   VAR_IN_OUT 
      xNewRecord { ExternalAccessible := 'False'; ExternalVisible := 'False'; ExternalWritable := 'False'} : Bool;
      xProductionRecord { ExternalAccessible := 'False'; ExternalVisible := 'False'; ExternalWritable := 'False'} : Bool;
      xLeftRobotUsed { ExternalAccessible := 'False'; ExternalVisible := 'False'; ExternalWritable := 'False'} : Bool;
      xRightRobotUsed { ExternalAccessible := 'False'; ExternalVisible := 'False'; ExternalWritable := 'False'} : Bool;
      xResetCurrentRecord { ExternalAccessible := 'False'; ExternalVisible := 'False'; ExternalWritable := 'False'} : Bool;
      xEraseAllData { ExternalAccessible := 'False'; ExternalVisible := 'False'; ExternalWritable := 'False'} : Bool;
      xDisplayNextRecord { ExternalAccessible := 'False'; ExternalVisible := 'False'; ExternalWritable := 'False'} : Bool;
      xDisplayPrevRecord { ExternalAccessible := 'False'; ExternalVisible := 'False'; ExternalWritable := 'False'} : Bool;
      uiNumberOfRecords { ExternalAccessible := 'False'; ExternalVisible := 'False'; ExternalWritable := 'False'} : UInt;
      aProdData : Array[*] of "stProductionRecord";
   END_VAR

   VAR 
      sxNewRecord { ExternalAccessible := 'False'; ExternalVisible := 'False'; ExternalWritable := 'False'} : Bool;
      sdiMaxRecord { ExternalAccessible := 'False'; ExternalVisible := 'False'; ExternalWritable := 'False'} : DInt;
      snCounter { ExternalAccessible := 'False'; ExternalVisible := 'False'; ExternalWritable := 'False'} : Int;
      suiMemDisplayCurentReccord { ExternalAccessible := 'False'; ExternalVisible := 'False'; ExternalWritable := 'False'} : UInt;
      suiMaxJobNumber { ExternalAccessible := 'False'; ExternalVisible := 'False'; ExternalWritable := 'False'} : UInt;
      suiMemCurrentJobNumberR1 { ExternalAccessible := 'False'; ExternalVisible := 'False'; ExternalWritable := 'False'} : UInt;
      suiMemCurrentJobNumberR2 { ExternalAccessible := 'False'; ExternalVisible := 'False'; ExternalWritable := 'False'} : UInt;
      suiDisplayCurentRecord { ExternalAccessible := 'False'; ExternalVisible := 'False'; ExternalWritable := 'False'} : UInt;
   END_VAR

   VAR_TEMP 
      txRequestAction : Bool;
      suiCount : UInt;
      suiRecord : UInt;
      tuiPaperUsedRobot1 : UInt;
      tuiPaperUsedRobot2 : UInt;
   END_VAR


BEGIN
	REGION Control Job Number Used
	  // Control if record data is in pregress and Job Data number change
	  IF #sxNewRecord AND (#uiCurrentJobNumberRobot1 <> #suiMemCurrentJobNumberR1) THEN
	    // Controo if job data number is in range
	    IF ((#uiCurrentJobNumberRobot1 > 0) AND (#uiCurrentJobNumberRobot1 <= 6)) THEN
	      #suiMemCurrentJobNumberR1 := #uiCurrentJobNumberRobot1;
	      CASE #uiCurrentJobNumberRobot1 OF
	        1:
	          #aProdData[1].Rob1Job1Used := TRUE;
	          #aProdData[1].Rob1Job1DistChangePaper := #WorkRecipe.RecipeLayerType.JobTableLeft[1].WornPaperDistance;
	          #aProdData[1].Rob1Job1ForceTarget := #WorkRecipe.RecipeLayerType.JobTableLeft[1].SetForceTarget;
	          #aProdData[1].Rob1Job1RobotSpeed := #WorkRecipe.RecipeLayerType.JobTableLeft[1].SetRobotSpeed;
	          #aProdData[1].Rob1Job1SandingSpeed := #WorkRecipe.RecipeLayerType.JobTableLeft[1].SetSpeed;
	        2:
	          #aProdData[1].Rob1Job2Used := TRUE;
	          #aProdData[1].Rob1Job2DistChangePaper := #WorkRecipe.RecipeLayerType.JobTableLeft[2].WornPaperDistance;
	          #aProdData[1].Rob1Job2ForceTarget := #WorkRecipe.RecipeLayerType.JobTableLeft[2].SetForceTarget;
	          #aProdData[1].Rob1Job2RobotSpeed := #WorkRecipe.RecipeLayerType.JobTableLeft[2].SetRobotSpeed;
	          #aProdData[1].Rob1Job2SandingSpeed := #WorkRecipe.RecipeLayerType.JobTableLeft[2].SetSpeed;
	        3:
	          #aProdData[1].Rob1Job3Used := TRUE;
	          #aProdData[1].Rob1Job3DistChangePaper := #WorkRecipe.RecipeLayerType.JobTableLeft[3].WornPaperDistance;
	          #aProdData[1].Rob1Job3ForceTarget := #WorkRecipe.RecipeLayerType.JobTableLeft[3].SetForceTarget;
	          #aProdData[1].Rob1Job3RobotSpeed := #WorkRecipe.RecipeLayerType.JobTableLeft[3].SetRobotSpeed;
	          #aProdData[1].Rob1Job3SandingSpeed := #WorkRecipe.RecipeLayerType.JobTableLeft[3].SetSpeed;
	        4:
	          #aProdData[1].Rob1Job4Used := TRUE;
	          #aProdData[1].Rob1Job4DistChangePaper := #WorkRecipe.RecipeLayerType.JobTableLeft[4].WornPaperDistance;
	          #aProdData[1].Rob1Job4ForceTarget := #WorkRecipe.RecipeLayerType.JobTableLeft[4].SetForceTarget;
	          #aProdData[1].Rob1Job4RobotSpeed := #WorkRecipe.RecipeLayerType.JobTableLeft[4].SetRobotSpeed;
	          #aProdData[1].Rob1Job4SandingSpeed := #WorkRecipe.RecipeLayerType.JobTableLeft[4].SetSpeed;
	        5:
	          #aProdData[1].Rob1Job5Used := TRUE;
	          #aProdData[1].Rob1Job5DistChangePaper := #WorkRecipe.RecipeLayerType.JobTableLeft[5].WornPaperDistance;
	          #aProdData[1].Rob1Job5ForceTarget := #WorkRecipe.RecipeLayerType.JobTableLeft[5].SetForceTarget;
	          #aProdData[1].Rob1Job5RobotSpeed := #WorkRecipe.RecipeLayerType.JobTableLeft[5].SetRobotSpeed;
	          #aProdData[1].Rob1Job5SandingSpeed := #WorkRecipe.RecipeLayerType.JobTableLeft[5].SetSpeed;
	        6:
	          #aProdData[1].Rob1Job6Used := TRUE;
	          #aProdData[1].Rob1Job6DistChangePaper := #WorkRecipe.RecipeLayerType.JobTableLeft[6].WornPaperDistance;
	          #aProdData[1].Rob1Job6ForceTarget := #WorkRecipe.RecipeLayerType.JobTableLeft[6].SetForceTarget;
	          #aProdData[1].Rob1Job6RobotSpeed := #WorkRecipe.RecipeLayerType.JobTableLeft[6].SetRobotSpeed;
	          #aProdData[1].Rob1Job6SandingSpeed := #WorkRecipe.RecipeLayerType.JobTableLeft[6].SetSpeed;
	      END_CASE;
	      
	    ELSE
	      #suiMemCurrentJobNumberR1 := #uiCurrentJobNumberRobot1;
	    END_IF;
	  END_IF;
	  
	  // Control if record data is in pregress and Job Data number change
	  IF #sxNewRecord AND (#uiCurrentJobNumberRobot2 <> #suiMemCurrentJobNumberR2) THEN
	    // Controo if job data number is in range
	    IF ((#uiCurrentJobNumberRobot2 > 0) AND (#uiCurrentJobNumberRobot2 <= 6)) THEN
	      #suiMemCurrentJobNumberR2 := #uiCurrentJobNumberRobot2;
	      CASE #uiCurrentJobNumberRobot2 OF
	        1:
	          #aProdData[1].Rob2Job1Used := TRUE;
	          #aProdData[1].Rob2Job1DistChangePaper := #WorkRecipe.RecipeLayerType.JobTableRight[1].WornPaperDistance;
	          #aProdData[1].Rob2Job1ForceTarget := #WorkRecipe.RecipeLayerType.JobTableRight[1].SetForceTarget;
	          #aProdData[1].Rob2Job1RobotSpeed := #WorkRecipe.RecipeLayerType.JobTableRight[1].SetRobotSpeed;
	          #aProdData[1].Rob2Job1SandingSpeed := #WorkRecipe.RecipeLayerType.JobTableRight[1].SetSpeed;
	        2:
	          #aProdData[1].Rob2Job2Used := TRUE;
	          #aProdData[1].Rob2Job2DistChangePaper := #WorkRecipe.RecipeLayerType.JobTableRight[2].WornPaperDistance;
	          #aProdData[1].Rob2Job2ForceTarget := #WorkRecipe.RecipeLayerType.JobTableRight[2].SetForceTarget;
	          #aProdData[1].Rob2Job2RobotSpeed := #WorkRecipe.RecipeLayerType.JobTableRight[2].SetRobotSpeed;
	          #aProdData[1].Rob2Job2SandingSpeed := #WorkRecipe.RecipeLayerType.JobTableRight[2].SetSpeed;
	        3:
	          #aProdData[1].Rob2Job3Used := TRUE;
	          #aProdData[1].Rob2Job3DistChangePaper := #WorkRecipe.RecipeLayerType.JobTableRight[3].WornPaperDistance;
	          #aProdData[1].Rob2Job3ForceTarget := #WorkRecipe.RecipeLayerType.JobTableRight[3].SetForceTarget;
	          #aProdData[1].Rob2Job3RobotSpeed := #WorkRecipe.RecipeLayerType.JobTableRight[3].SetRobotSpeed;
	          #aProdData[1].Rob2Job3SandingSpeed := #WorkRecipe.RecipeLayerType.JobTableRight[3].SetSpeed;
	        4:
	          #aProdData[1].Rob2Job4Used := TRUE;
	          #aProdData[1].Rob2Job4DistChangePaper := #WorkRecipe.RecipeLayerType.JobTableRight[4].WornPaperDistance;
	          #aProdData[1].Rob2Job4ForceTarget := #WorkRecipe.RecipeLayerType.JobTableRight[4].SetForceTarget;
	          #aProdData[1].Rob2Job4RobotSpeed := #WorkRecipe.RecipeLayerType.JobTableRight[4].SetRobotSpeed;
	          #aProdData[1].Rob2Job4SandingSpeed := #WorkRecipe.RecipeLayerType.JobTableRight[4].SetSpeed;
	        5:
	          #aProdData[1].Rob2Job5Used := TRUE;
	          #aProdData[1].Rob2Job5DistChangePaper := #WorkRecipe.RecipeLayerType.JobTableRight[5].WornPaperDistance;
	          #aProdData[1].Rob2Job5ForceTarget := #WorkRecipe.RecipeLayerType.JobTableRight[5].SetForceTarget;
	          #aProdData[1].Rob2Job5RobotSpeed := #WorkRecipe.RecipeLayerType.JobTableRight[5].SetRobotSpeed;
	          #aProdData[1].Rob2Job5SandingSpeed := #WorkRecipe.RecipeLayerType.JobTableRight[5].SetSpeed;
	        6:
	          #aProdData[1].Rob2Job6Used := TRUE;
	          #aProdData[1].Rob2Job6DistChangePaper := #WorkRecipe.RecipeLayerType.JobTableRight[6].WornPaperDistance;
	          #aProdData[1].Rob2Job6ForceTarget := #WorkRecipe.RecipeLayerType.JobTableRight[6].SetForceTarget;
	          #aProdData[1].Rob2Job6RobotSpeed := #WorkRecipe.RecipeLayerType.JobTableRight[6].SetRobotSpeed;
	          #aProdData[1].Rob2Job6SandingSpeed := #WorkRecipe.RecipeLayerType.JobTableRight[6].SetSpeed;
	      END_CASE;
	    ELSE
	      #suiMemCurrentJobNumberR2 := #uiCurrentJobNumberRobot2;
	    END_IF;
	  END_IF;
	END_REGION
	
	REGION Exit FB
	  // Exit function bloc if no action requested
	  IF #suiDisplayCurentRecord = 0 THEN
	    #suiDisplayCurentRecord := 1;
	  END_IF;
	  
	  #txRequestAction := #xNewRecord OR #xProductionRecord OR #xResetCurrentRecord OR #xEraseAllData OR #xDisplayNextRecord OR #xDisplayPrevRecord;
	  IF #suiDisplayCurentRecord <> #suiMemDisplayCurentReccord THEN
	    #suiMemDisplayCurentReccord := #suiDisplayCurentRecord;
	  ELSIF (NOT #txRequestAction) THEN
	    RETURN;
	  END_IF;
	END_REGION
	
	REGION Record Min and Max
	  #sdiMaxRecord := UPPER_BOUND(ARR := #aProdData, DIM := 1);
	  IF #uiNumberOfRecords < 1 THEN
	    #uiRecordMax := 1;
	  ELSE
	    #uiRecordMax := #uiNumberOfRecords;
	  END_IF;
	  #uiRecordMin := 1;
	END_REGION
	
	REGION New Record
	  IF #xNewRecord AND (NOT #sxNewRecord) THEN // Request new record and no new record in progress
	    IF #uiNumberOfRecords = 0 THEN // First record
	      // First record in the table
	      #uiNumberOfRecords := 1;
	      // Erase all data
	      #aProdData[1] := #aProdData[0];
	      "FC71_PrepareNewRecord"(usiCurrentLayerType:=#usiCurrentLayerType,
	                              uiCbsNumber:=#uiCbsNumber,
	                              WorkRecipe:=#WorkRecipe,
	                              ProdData:=#aProdData[1]);
	    ELSIF #uiNumberOfRecords < #sdiMaxRecord THEN // less then max record
	      // Increase the number of record
	      #uiNumberOfRecords += 1;
	      // Offset all records
	      FOR #snCounter := UINT_TO_INT(#uiNumberOfRecords) TO 2 BY -1 DO
	        #aProdData[#snCounter] := #aProdData[#snCounter - 1];
	      END_FOR;
	      // Erase all data
	      #aProdData[1] := #aProdData[0];
	      "FC71_PrepareNewRecord"(usiCurrentLayerType := #usiCurrentLayerType,
	                              uiCbsNumber := #uiCbsNumber,
	                              WorkRecipe := #WorkRecipe,
	                              ProdData := #aProdData[1]);
	    ELSIF #uiNumberOfRecords = #sdiMaxRecord THEN // Max record
	      // Delete last record
	      #aProdData[#uiNumberOfRecords] := #aProdData[0];
	      // Offset all records
	      FOR #snCounter := UINT_TO_INT(#uiNumberOfRecords) TO 2 BY -1 DO
	        #aProdData[#snCounter] := #aProdData[#snCounter - 1];
	      END_FOR;
	      // Erase all data
	      #aProdData[1] := #aProdData[0];
	      "FC71_PrepareNewRecord"(usiCurrentLayerType := #usiCurrentLayerType,
	                              uiCbsNumber := #uiCbsNumber,
	                              WorkRecipe := #WorkRecipe,
	                              ProdData := #aProdData[1]);
	    END_IF;
	    #xNewRecord := FALSE;
	    #sxNewRecord := TRUE;
	    
	  ELSIF #xNewRecord AND #sxNewRecord THEN // Request new record but new record already in progress
	    #xNewRecord := FALSE;
	  END_IF;
	END_REGION
	
	REGION Production Record
	  IF #xProductionRecord AND #sxNewRecord THEN // Request record production and new record already in progress
	    // Count paper used if robot 1 used
	    IF #xLeftRobotUsed THEN
	      #tuiPaperUsedRobot1 := #uiPaperUsedRobot1;
	      #xLeftRobotUsed := FALSE;
	    ELSE
	      #tuiPaperUsedRobot1 := 0;
	    END_IF;
	    // Count paper used if robot 2 used
	    IF #xRightRobotUsed THEN
	      #tuiPaperUsedRobot2 := #uiPaperUsedRobot2;
	      #xRightRobotUsed := FALSE;
	    ELSE
	      #tuiPaperUsedRobot2 := 0;
	    END_IF;
	    // General record
	    "FC72_Record"(uiPaperUsedRobot1:=#tuiPaperUsedRobot1,
	                  uiPaperUsedRobot2:=#tuiPaperUsedRobot2,
	                  ProdData:=#aProdData[1]);
	    
	    #xProductionRecord := FALSE;
	    #sxNewRecord := FALSE;
	    
	  ELSIF #xProductionRecord AND (NOT #sxNewRecord) THEN // Request record production but no new record already in progress
	    #xProductionRecord := FALSE;
	    
	  END_IF;
	END_REGION
	
	REGION Erase All
	  IF #xEraseAllData THEN // Request reset all record in the table
	    // Erase all the data record
	    FOR #snCounter := 1 TO UINT_TO_INT(#uiNumberOfRecords) DO
	      #aProdData[#snCounter] := #aProdData[0];
	    END_FOR;
	    // Reset the number of record in table
	    #suiDisplayCurentRecord := 1;
	    #uiNumberOfRecords := 0;
	    #sxNewRecord := FALSE;
	    #xEraseAllData := FALSE;
	  END_IF;
	END_REGION
	
	REGION Erase Record
	  IF #xResetCurrentRecord AND #sxNewRecord THEN // Request reset current record and new record already in progress
	    // Offset all current record down
	    FOR #snCounter := 1 TO (UINT_TO_INT(#uiNumberOfRecords) - 1) DO
	      #aProdData[#snCounter] := #aProdData[#snCounter + 1];
	    END_FOR;
	    // Erase the last record in the table
	    #aProdData[#uiNumberOfRecords] := #aProdData[0];
	    // Decrease the number of records in the table
	    #uiNumberOfRecords -= 1;
	    #sxNewRecord := FALSE;
	    #xResetCurrentRecord := FALSE;
	    
	  ELSIF #xResetCurrentRecord AND (NOT #sxNewRecord) THEN // Request reset current record but no new record already in progress
	    #xResetCurrentRecord := FALSE;
	  END_IF;
	END_REGION
	
	REGION change curent record displayed
	  // Force display current record to 1
	  IF #suiDisplayCurentRecord = 0 THEN
	    #suiDisplayCurentRecord := 1;
	  END_IF;
	  
	  // Increase curent displayed record number
	  IF #xDisplayNextRecord AND (#uiRecordMax >= (#suiDisplayCurentRecord + 10)) THEN
	    #suiDisplayCurentRecord += 10;
	    #xDisplayNextRecord := FALSE;
	  ELSE
	    #xDisplayNextRecord := FALSE;
	  END_IF;
	  
	  // Decrease current displayed record number
	  IF #xDisplayPrevRecord AND (#suiDisplayCurentRecord > #uiRecordMin) THEN
	    #suiDisplayCurentRecord -= 10;
	    #xDisplayPrevRecord := FALSE;
	  ELSE
	    #xDisplayPrevRecord := FALSE;
	  END_IF;
	  
	  
	END_REGION
	
	REGION Refresh displayed record
	  #uiNbrDisplyedLine := 0;
	  #uiFirstRecordDisplayed := 0;
	  #uiLastRecordDisplayed := 0;
	  IF (#suiDisplayCurentRecord <= #uiRecordMax) AND (#uiNumberOfRecords <> 0) THEN
	    #uiNbrDisplyedLine += 1;
	    #uiFirstRecordDisplayed := #suiDisplayCurentRecord;
	    #uiLastRecordDisplayed := #suiDisplayCurentRecord;
	    #aDisplayProdData[0] := #aProdData[#suiDisplayCurentRecord];
	  END_IF;
	  FOR #suiCount := 1 TO 9 DO
	    #suiRecord := (#suiDisplayCurentRecord + #suiCount);
	    IF #suiRecord <= #uiRecordMax THEN
	      #uiNbrDisplyedLine += 1;
	      #uiLastRecordDisplayed := #suiRecord;
	      #aDisplayProdData[#suiCount] := #aProdData[#suiRecord];
	    END_IF;
	  END_FOR;
	  #suiMemDisplayCurentReccord := #suiDisplayCurentRecord;
	  
	END_REGION
END_FUNCTION_BLOCK

FUNCTION "FC71_PrepareNewRecord" : Void
{ S7_Optimized_Access := 'TRUE' }
VERSION : 0.1
   VAR_INPUT 
      usiCurrentLayerType : USInt;
      uiCbsNumber : UInt;
      WorkRecipe : "stWorkRecipe";
   END_VAR

   VAR_IN_OUT 
      ProdData : "stProductionRecord";
   END_VAR

   VAR_TEMP 
      tdtlLocal {InstructionName := 'DTL'; LibVersion := '1.0'} : DTL;
      tnReturnValue : Int;
      tnCounter : Int;
   END_VAR


BEGIN
	// Read local date and time
	#tnReturnValue := RD_LOC_T(OUT => #tdtlLocal);
	// Reccord current date
	#ProdData.dDate := DTL_TO_DATE(#tdtlLocal);
	// Record current time
	#ProdData.todTime := DTL_TO_TOD(#tdtlLocal);
	// Record Name and Layer production
	#ProdData.sRecipeName := #WorkRecipe.RecipeName;
	#ProdData.sRecipeLayerTypeName := #WorkRecipe.RecipeLayerType.RecipeLayerTypeName;
	// Record Prog Number and layer type number
	#ProdData.usiProgNumber := #WorkRecipe.RecipeTrajNumber;
	#ProdData.usiLayerTypeNumber := #usiCurrentLayerType;
	// Record CBS serial Number
	#ProdData.uiCbsNumber := #uiCbsNumber;
	//Reset all job data
	(* // already done by copy ProdData[0] in ProdData[1]
	FOR #tnCounter := 1 TO 6 DO
	  // Job data for robot 1
	  #ProdData.JobRobot1[#tnCounter].JobUsed := FALSE;
	  #ProdData.JobRobot1[#tnCounter].DistanceChangePaper := 0;
	  #ProdData.JobRobot1[#tnCounter].ForceTarget := 0;
	  #ProdData.JobRobot1[#tnCounter].RobotSpeed := 0;
	  #ProdData.JobRobot1[#tnCounter].SandingSpeed := 0;
	  // Jod data for robot 2
	  #ProdData.JobRobot2[#tnCounter].JobUsed := FALSE;
	  #ProdData.JobRobot2[#tnCounter].DistanceChangePaper := 0;
	  #ProdData.JobRobot2[#tnCounter].ForceTarget := 0;
	  #ProdData.JobRobot2[#tnCounter].RobotSpeed := 0;
	  #ProdData.JobRobot2[#tnCounter].SandingSpeed := 0;
	END_FOR;
	*)
END_FUNCTION

FUNCTION "FC72_Record" : Void
{ S7_Optimized_Access := 'TRUE' }
VERSION : 0.1
   VAR_INPUT 
      uiPaperUsedRobot1 : UInt;
      uiPaperUsedRobot2 : UInt;
   END_VAR

   VAR_IN_OUT 
      ProdData : "stProductionRecord";
   END_VAR

   VAR_TEMP 
      tdtlLocal {InstructionName := 'DTL'; LibVersion := '1.0'} : DTL;
      tnReturnValue : Int;
      tdDate : Date;
      ttodTime : Time_Of_Day;
      tdiRecordTime : DInt;
      tdiMaxTime : DInt;
      tdiCurrentTime : DInt;
      tdiTemp : DInt;
   END_VAR

   VAR CONSTANT 
      ctodMaxTime : Time_Of_Day := TOD#23:59:59;
   END_VAR


BEGIN
	// Read local date and time
	#tnReturnValue := RD_LOC_T(OUT => #tdtlLocal);
	#tdDate := DTL_TO_DATE(#tdtlLocal);
	#ttodTime := DTL_TO_TOD(#tdtlLocal);
	
	// Control if same day or next day
	IF #tdDate <> #ProdData.dDate THEN
	  #tdiRecordTime := TOD_TO_DINT(#ProdData.todTime);
	  #tdiCurrentTime := TOD_TO_DINT(#ttodTime);
	  #tdiMaxTime := TOD_TO_DINT(#ProdData.todTime);
	  #tdiTemp := (#tdiMaxTime - #tdiRecordTime) + #tdiCurrentTime;
	  
	ELSE
	  #tdiRecordTime := TOD_TO_DINT(#ProdData.todTime);
	  #tdiCurrentTime := TOD_TO_DINT(#ttodTime);
	  #tdiTemp := (#tdiCurrentTime - #tdiRecordTime);
	  
	END_IF;
	
	#ProdData.tCycleTime := DINT_TO_TOD(#tdiTemp);
	
	#ProdData.uiPaperUsed := #uiPaperUsedRobot1 + #uiPaperUsedRobot2;
END_FUNCTION

FUNCTION_BLOCK "FB71_FlatnessCtrlRecord"
{ S7_Optimized_Access := 'TRUE' }
VERSION : 0.1
   VAR_OUTPUT 
      uiRecordMax { ExternalAccessible := 'False'; ExternalVisible := 'False'; ExternalWritable := 'False'} : UInt;
      uiRecordMin { ExternalAccessible := 'False'; ExternalVisible := 'False'; ExternalWritable := 'False'} : UInt;
      DisplayFlatRecData { ExternalAccessible := 'False'; ExternalVisible := 'False'; ExternalWritable := 'False'} : "stFlatnessCtrlRecord";
   END_VAR

   VAR_IN_OUT 
      xEraseAllData { ExternalAccessible := 'False'; ExternalVisible := 'False'; ExternalWritable := 'False'} : Bool;
      xDisplayNextRecord { ExternalAccessible := 'False'; ExternalVisible := 'False'; ExternalWritable := 'False'} : Bool;
      xDisplayPrevRecord { ExternalAccessible := 'False'; ExternalVisible := 'False'; ExternalWritable := 'False'} : Bool;
      uiDisplayCurentRecord { ExternalAccessible := 'False'; ExternalVisible := 'False'; ExternalWritable := 'False'} : UInt;
      uiNumberOfRecords { ExternalAccessible := 'False'; ExternalVisible := 'False'; ExternalWritable := 'False'} : UInt;
      stFlatnessdata : "stFlatnessData";
      aFlatnessData : Array[*] of "stFlatnessCtrlRecord";
   END_VAR

   VAR 
      sdiMaxRecord { ExternalAccessible := 'False'; ExternalVisible := 'False'; ExternalWritable := 'False'} : DInt;
      siCounter { ExternalAccessible := 'False'; ExternalVisible := 'False'; ExternalWritable := 'False'} : Int;
      suiMemDisplayCurentReccord { ExternalAccessible := 'False'; ExternalVisible := 'False'; ExternalWritable := 'False'} : UInt;
   END_VAR

   VAR_TEMP 
      tiReturnValue : Int;
      tdtlActualDateTime {InstructionName := 'DTL'; LibVersion := '1.0'} : DTL;
   END_VAR


BEGIN
	// Exit function bloc if no action requested
	IF #uiDisplayCurentRecord = 0 THEN
	  #uiDisplayCurentRecord := 1;
	END_IF;
	
	IF (NOT #stFlatnessdata.xFlatnessCrtlRequestRecord) AND #stFlatnessdata.xFlatnessCtrlRecorded THEN
	  #stFlatnessdata.xFlatnessCtrlRecorded := FALSE;
	  RETURN;
	ELSIF #uiDisplayCurentRecord <> #suiMemDisplayCurentReccord THEN
	  #suiMemDisplayCurentReccord := #uiDisplayCurentRecord;
	ELSIF ((NOT #stFlatnessdata.xFlatnessCrtlRequestRecord) OR #stFlatnessdata.xFlatnessCtrlRecorded) AND (NOT #xEraseAllData) AND (NOT #xDisplayNextRecord) AND (NOT #xDisplayPrevRecord) THEN
	  RETURN;
	END_IF;
	
	REGION Record Min and Max
	  #sdiMaxRecord := UPPER_BOUND(ARR := #aFlatnessData, DIM := 1);
	  IF #uiNumberOfRecords < 1 THEN
	    #uiRecordMax := 1;
	  ELSE
	    #uiRecordMax := #uiNumberOfRecords;
	  END_IF;
	  #uiRecordMin := 1;
	END_REGION
	
	
	
	REGION Erase All Data
	  IF #xEraseAllData THEN
	    // Erase all the data record
	    FOR #siCounter := 1 TO UINT_TO_INT(#uiNumberOfRecords) DO
	      #aFlatnessData[#siCounter] := #aFlatnessData[0];
	    END_FOR;
	    // Reset the number of record in table
	    #uiDisplayCurentRecord := 1;
	    #uiNumberOfRecords := 0;
	    #xEraseAllData := FALSE;
	  END_IF;
	END_REGION
	
	REGION Flatness Record data
	  IF #stFlatnessdata.xFlatnessCrtlRequestRecord THEN
	    
	    IF #uiNumberOfRecords = 0 THEN // First record
	      // First record in the table
	      #uiNumberOfRecords := 1;
	    ELSIF #uiNumberOfRecords < #sdiMaxRecord THEN // less then max record
	      // Increase the number of record
	      #uiNumberOfRecords += 1;
	      // Offset all records
	      FOR #siCounter := UINT_TO_INT(#uiNumberOfRecords) TO 2 BY -1 DO
	        #aFlatnessData[#siCounter] := #aFlatnessData[#siCounter - 1];
	      END_FOR;
	    ELSIF #uiNumberOfRecords = #sdiMaxRecord THEN // Max record
	      // Delete last record
	      #aFlatnessData[#uiNumberOfRecords] := #aFlatnessData[0];
	      // Offset all records
	      FOR #siCounter := UINT_TO_INT(#uiNumberOfRecords) TO 2 BY -1 DO
	        #aFlatnessData[#siCounter] := #aFlatnessData[#siCounter - 1];
	      END_FOR;
	    END_IF;
	    
	    #tiReturnValue := RD_LOC_T(#tdtlActualDateTime);
	    #aFlatnessData[1].dtlDataTime := #tdtlActualDateTime;
	    #aFlatnessData[1].xFlatnessResult := #stFlatnessdata.xFlatnessCtrlPassed;
	    #aFlatnessData[1].uiStrokePositionDiskA := #stFlatnessdata.uiStrokePositionDiskA;
	    #aFlatnessData[1].uiStrokePositionDiskB := #stFlatnessdata.uiStrokePositionDiskB;
	    #aFlatnessData[1].uiStrokePositionDiskC := #stFlatnessdata.uiStrokePositionDiskC;
	    
	    #stFlatnessdata.xFlatnessCtrlRecorded := true;
	    
	  END_IF;
	END_REGION
	
	
	REGION change curent record displayed
	  // Increase curent displayed record number
	  IF #xDisplayNextRecord AND (#uiDisplayCurentRecord < #uiRecordMax) THEN
	    #uiDisplayCurentRecord += 1;
	    #xDisplayNextRecord := FALSE;
	  ELSE
	    #xDisplayNextRecord := FALSE;
	  END_IF;
	  
	  // Decrease current displayed record number
	  IF #xDisplayPrevRecord AND (#uiDisplayCurentRecord > #uiRecordMin) THEN
	    #uiDisplayCurentRecord -= 1;
	    #xDisplayPrevRecord := FALSE;
	  ELSE
	    #xDisplayPrevRecord := FALSE;
	  END_IF;
	  
	  
	END_REGION
	
	REGION Refresh displayed record
	  
	  #DisplayFlatRecData := #aFlatnessData[#uiDisplayCurentRecord];
	  #suiMemDisplayCurentReccord := #uiDisplayCurentRecord;
	  
	END_REGION
	
	
END_FUNCTION_BLOCK

FUNCTION "FC80_TeepTrack" : Void   // FC80, LAD
{ S7_Optimized_Access := 'TRUE' }
// stored: AutoNumber false, SetENOAutomatically false
BEGIN

REGION Network 1: Teep Track Robot 1
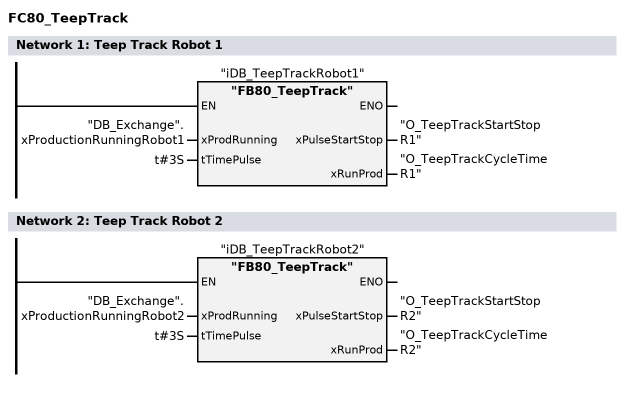
   RUNG wire#powerrail
      "iDB_TeepTrackRobot1"(xProdRunning := "DB_Exchange".xProductionRunningRobot1, tTimePulse := t#3S, xPulseStartStop => "O_TeepTrackStartStopR1", xRunProd => "O_TeepTrackCycleTimeR1")
   END_RUNG
   // the same network as SCL:
   "iDB_TeepTrackRobot1"(xProdRunning := "DB_Exchange".xProductionRunningRobot1,   // "FB80_TeepTrack"
                         tTimePulse := t#3S,
                         xPulseStartStop => "O_TeepTrackStartStopR1",
                         xRunProd => "O_TeepTrackCycleTimeR1");
END_REGION

REGION Network 2: Teep Track Robot 2
   RUNG wire#powerrail
      "iDB_TeepTrackRobot2"(xProdRunning := "DB_Exchange".xProductionRunningRobot2, tTimePulse := t#3S, xPulseStartStop => "O_TeepTrackStartStopR2", xRunProd => "O_TeepTrackCycleTimeR2")
   END_RUNG
   // the same network as SCL:
   "iDB_TeepTrackRobot2"(xProdRunning := "DB_Exchange".xProductionRunningRobot2,   // "FB80_TeepTrack"
                         tTimePulse := t#3S,
                         xPulseStartStop => "O_TeepTrackStartStopR2",
                         xRunProd => "O_TeepTrackCycleTimeR2");
END_REGION
END_FUNCTION

FUNCTION_BLOCK "FB80_TeepTrack"   // FB80, LAD
{ S7_Optimized_Access := 'TRUE' }
// stored: AutoNumber false, MemoryReserve 100, SetENOAutomatically false
   VAR_INPUT
      xProdRunning { ExternalAccessible := 'False'; ExternalVisible := 'False'; ExternalWritable := 'False'} : Bool;   // Production Running
      tTimePulse { ExternalAccessible := 'False'; ExternalVisible := 'False'; ExternalWritable := 'False'} : Time;   // Time for pulse StartStop
   END_VAR
   VAR_OUTPUT
      xPulseStartStop { ExternalAccessible := 'False'; ExternalVisible := 'False'; ExternalWritable := 'False'} : Bool;   // Pulse Start stop
      xRunProd { ExternalAccessible := 'False'; ExternalVisible := 'False'; ExternalWritable := 'False'} : Bool;   // Production running
   END_VAR
   VAR
      sxMemRun { ExternalAccessible := 'False'; ExternalVisible := 'False'; ExternalWritable := 'False'} : Bool;
      miDB_PulseStartStop { ExternalAccessible := 'False'; ExternalVisible := 'False'; ExternalWritable := 'False'; S7_SetPoint := 'True'} : TP_TIME;
      sxFPMemRun { ExternalAccessible := 'False'; ExternalVisible := 'False'; ExternalWritable := 'False'} : Bool;
      sxFNMemRun { ExternalAccessible := 'False'; ExternalVisible := 'False'; ExternalWritable := 'False'} : Bool;
   END_VAR
   VAR_TEMP   // added for the SCL form of the ladder/FBD networks
      _w1 : Bool;
      _w2 : Bool;
   END_VAR
BEGIN

REGION Network 1: Production running
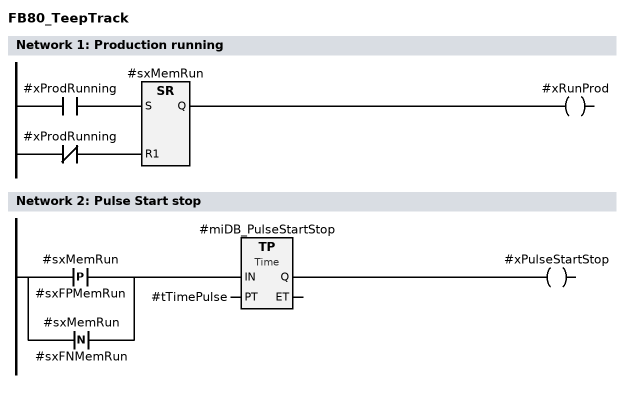
   RUNG wire#powerrail
      Contact( #xProdRunning )
      S_SR(operand := #sxMemRun, r1 := wire#w1)
      Coil( #xRunProd )
   END_RUNG
   RUNG wire#powerrail
      I_Contact( #xProdRunning )
   END_RUNG wire#w1
   // the same network as SCL:
   IF #xProdRunning THEN
       #sxMemRun := TRUE;   // SR flip-flop
   END_IF;
   IF NOT #xProdRunning THEN #sxMemRun := FALSE; END_IF;
   #xRunProd := #sxMemRun;
END_REGION

REGION Network 2: Pulse Start stop
   RUNG wire#powerrail
      P_Contact(operand := #sxMemRun, bit := #sxFPMemRun)
      wire#w1
      { S7_Templates := "time_type := Time" } #miDB_PulseStartStop.TP(pt := #tTimePulse, et =>)
      Coil( #xPulseStartStop )
   END_RUNG
   RUNG wire#powerrail
      N_Contact(operand := #sxMemRun, bit := #sxFNMemRun)
   END_RUNG wire#w1
   // the same network as SCL:
   #_w1 := #sxMemRun AND NOT #sxFPMemRun;   // rising edge of #sxMemRun
   #sxFPMemRun := #sxMemRun;
   #_w2 := NOT #sxMemRun AND #sxFNMemRun;   // falling edge of #sxMemRun
   #sxFNMemRun := #sxMemRun;
   #miDB_PulseStartStop(IN := #_w1 OR #_w2, PT := #tTimePulse);   // TP
   #xPulseStartStop := #miDB_PulseStartStop.Q;
END_REGION
END_FUNCTION_BLOCK

FUNCTION "FC90_SentronComm" : Void   // FC90, LAD
{ S7_Optimized_Access := 'TRUE' }
// stored: AutoNumber false, IsIECCheckEnabled true, SetENOAutomatically false
BEGIN

REGION Network 1: Read Sentron Main cabinet
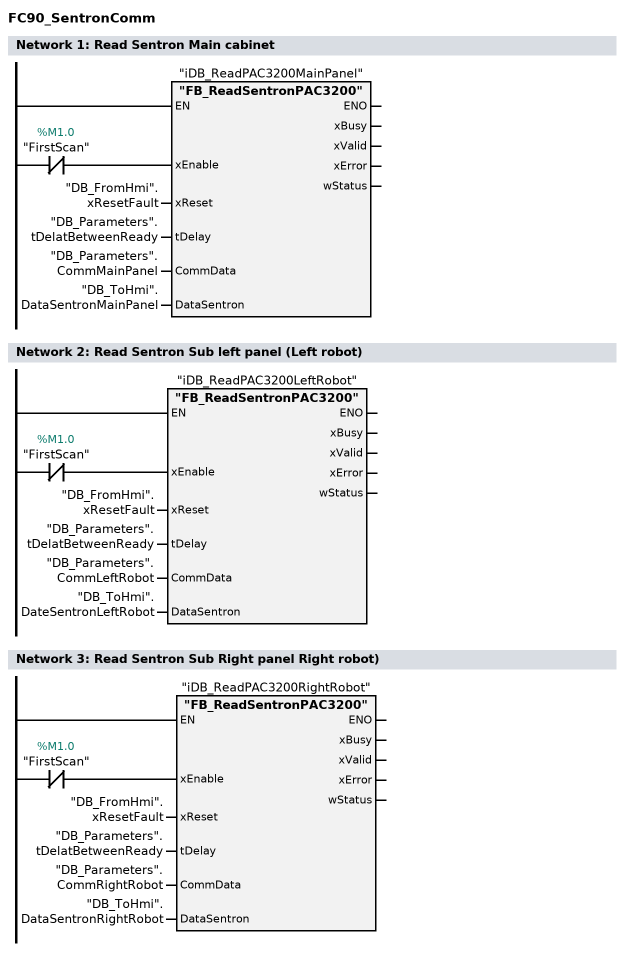
   RUNG wire#powerrail
      "iDB_ReadPAC3200MainPanel"(xEnable := wire#w1, xReset := "DB_FromHmi".xResetFault, tDelay := "DB_Parameters".tDelatBetweenReady, CommData := "DB_Parameters".CommMainPanel, DataSentron := "DB_ToHmi".DataSentronMainPanel, xBusy =>, xValid =>, xError =>, wStatus =>)
   END_RUNG
   RUNG wire#powerrail
      I_Contact( "FirstScan" )
   END_RUNG wire#w1
   // the same network as SCL:
   "iDB_ReadPAC3200MainPanel"(xEnable := NOT "FirstScan",   // "FB_ReadSentronPAC3200"
                           xReset := "DB_FromHmi".xResetFault,
                           tDelay := "DB_Parameters".tDelatBetweenReady,
                           CommData := "DB_Parameters".CommMainPanel,
                           DataSentron := "DB_ToHmi".DataSentronMainPanel);
END_REGION

REGION Network 2: Read Sentron Sub left panel (Left robot)
   RUNG wire#powerrail
      "iDB_ReadPAC3200LeftRobot"(xEnable := wire#w1, xReset := "DB_FromHmi".xResetFault, tDelay := "DB_Parameters".tDelatBetweenReady, CommData := "DB_Parameters".CommLeftRobot, DataSentron := "DB_ToHmi".DateSentronLeftRobot, xBusy =>, xValid =>, xError =>, wStatus =>)
   END_RUNG
   RUNG wire#powerrail
      I_Contact( "FirstScan" )
   END_RUNG wire#w1
   // the same network as SCL:
   "iDB_ReadPAC3200LeftRobot"(xEnable := NOT "FirstScan",   // "FB_ReadSentronPAC3200"
                           xReset := "DB_FromHmi".xResetFault,
                           tDelay := "DB_Parameters".tDelatBetweenReady,
                           CommData := "DB_Parameters".CommLeftRobot,
                           DataSentron := "DB_ToHmi".DateSentronLeftRobot);
END_REGION

REGION Network 3: Read Sentron Sub Right panel Right robot)
   RUNG wire#powerrail
      "iDB_ReadPAC3200RightRobot"(xEnable := wire#w1, xReset := "DB_FromHmi".xResetFault, tDelay := "DB_Parameters".tDelatBetweenReady, CommData := "DB_Parameters".CommRightRobot, DataSentron := "DB_ToHmi".DataSentronRightRobot, xBusy =>, xValid =>, xError =>, wStatus =>)
   END_RUNG
   RUNG wire#powerrail
      I_Contact( "FirstScan" )
   END_RUNG wire#w1
   // the same network as SCL:
   "iDB_ReadPAC3200RightRobot"(xEnable := NOT "FirstScan",   // "FB_ReadSentronPAC3200"
                           xReset := "DB_FromHmi".xResetFault,
                           tDelay := "DB_Parameters".tDelatBetweenReady,
                           CommData := "DB_Parameters".CommRightRobot,
                           DataSentron := "DB_ToHmi".DataSentronRightRobot);
END_REGION
END_FUNCTION

FUNCTION_BLOCK "FB_ReadSentronPAC3200"
{ S7_Optimized_Access := 'TRUE' }
VERSION : 0.1
   VAR_INPUT 
      xEnable { ExternalAccessible := 'False'; ExternalVisible := 'False'; ExternalWritable := 'False'} : Bool;   // Activation du bloc
      xReset { ExternalAccessible := 'False'; ExternalVisible := 'False'; ExternalWritable := 'False'} : Bool;
      tDelay { ExternalAccessible := 'False'; ExternalVisible := 'False'; ExternalWritable := 'False'} : Time;
      CommData {InstructionName := 'TCON_IP_v4'; LibVersion := '1.0'; ExternalAccessible := 'False'; ExternalVisible := 'False'; ExternalWritable := 'False'} : TCON_IP_v4;
   END_VAR

   VAR_OUTPUT 
      xBusy { ExternalAccessible := 'False'; ExternalVisible := 'False'; ExternalWritable := 'False'} : Bool;
      xValid { ExternalAccessible := 'False'; ExternalVisible := 'False'; ExternalWritable := 'False'} : Bool;
      xError { ExternalAccessible := 'False'; ExternalVisible := 'False'; ExternalWritable := 'False'} : Bool;
      wStatus { ExternalAccessible := 'False'; ExternalVisible := 'False'; ExternalWritable := 'False'} : Word;
   END_VAR

   VAR_IN_OUT 
      DataSentron : "Sentron_PAC";
   END_VAR

   VAR 
      swStatus { ExternalAccessible := 'False'; ExternalVisible := 'False'; ExternalWritable := 'False'} : Word := #StatusNoCall;
      sdiFbState { ExternalAccessible := 'False'; ExternalVisible := 'False'; ExternalWritable := 'False'} : DInt := #FB_StateNoProcessing;
      snStep { ExternalAccessible := 'False'; ExternalVisible := 'False'; ExternalWritable := 'False'} : Int;
      sxStartDelay { ExternalAccessible := 'False'; ExternalVisible := 'False'; ExternalWritable := 'False'} : Bool;
      sxValid { ExternalAccessible := 'False'; ExternalVisible := 'False'; ExternalWritable := 'False'} : Bool;
      sxBusy { ExternalAccessible := 'False'; ExternalVisible := 'False'; ExternalWritable := 'False'} : Bool;
      sxError { ExternalAccessible := 'False'; ExternalVisible := 'False'; ExternalWritable := 'False'} : Bool;
      sxErrorUserCleared { ExternalAccessible := 'False'; ExternalVisible := 'False'; ExternalWritable := 'False'} : Bool;
      sxErrorAutoCleared { ExternalAccessible := 'False'; ExternalVisible := 'False'; ExternalWritable := 'False'} : Bool;
      sxDisablingCompleted { ExternalAccessible := 'False'; ExternalVisible := 'False'; ExternalWritable := 'False'} : Bool;
      sxEnabledOld { ExternalAccessible := 'False'; ExternalVisible := 'False'; ExternalWritable := 'False'} : Bool;
      sxMBcReq { ExternalAccessible := 'False'; ExternalVisible := 'False'; ExternalWritable := 'False'} : Bool;
      sxMBcDisconnect { ExternalAccessible := 'False'; ExternalVisible := 'False'; ExternalWritable := 'False'} : Bool;
      sxMBcDone { ExternalAccessible := 'False'; ExternalVisible := 'False'; ExternalWritable := 'False'} : Bool;
      sxMBcBusy { ExternalAccessible := 'False'; ExternalVisible := 'False'; ExternalWritable := 'False'} : Bool;
      sxMBcError { ExternalAccessible := 'False'; ExternalVisible := 'False'; ExternalWritable := 'False'} : Bool;
      swMBcStatus { ExternalAccessible := 'False'; ExternalVisible := 'False'; ExternalWritable := 'False'} : Word;
      sudiMBcAddress { ExternalAccessible := 'False'; ExternalVisible := 'False'; ExternalWritable := 'False'} : UDInt;
      suiMBcLen { ExternalAccessible := 'False'; ExternalVisible := 'False'; ExternalWritable := 'False'} : UInt;
      sarDataTemp { ExternalAccessible := 'False'; ExternalVisible := 'False'; ExternalWritable := 'False'} : Array[0..34] of Real;
      miDB_ModbusClient {InstructionName := 'MB_CLIENT'; LibVersion := '6.0'; ExternalAccessible := 'False'; ExternalVisible := 'False'; ExternalWritable := 'False'} : MB_CLIENT;
      miDB_TonDelay {InstructionName := 'TON_TIME'; LibVersion := '1.0'; ExternalAccessible := 'False'; ExternalVisible := 'False'; ExternalWritable := 'False'} : TON_TIME;
   END_VAR

   VAR_TEMP 
      txEnable : Bool;
   END_VAR

   VAR CONSTANT 
      FB_StateNoProcessing : DInt := 0;
      FB_StateEnabling : DInt := 10;
      FB_StateProcessing : DInt := 50;
      FB_StateDisabling : DInt := 90;
      StepInitial : Int := 0;
      StepReqPhase1 : Int := 10;
      StepWaitDonePh1 : Int := 20;
      StepWriteDataPh1 : Int := 40;
      StepReqPhase2 : Int := 50;
      StepWaitDonePh2 : Int := 60;
      StepWriteDataPh2 : Int := 80;
      StepReqPhase3 : Int := 90;
      StepWaitDonePh3 : Int := 100;
      StepWriteDataPh3 : Int := 120;
      StepWaitDelay : Int := 130;
      StatusNoCall : Word := 16#7000;
      StatusFirstCall : Word := 16#7001;
      StatusSubsequenceCall : Word := 16#7002;
      ErrUndefinedState : Word := 16#8600;
      ErrInBlocOperation : Word := 16#8001;
      ErrParametrization : Word := 16#8200;
      ErrProcessingExtern : Word := 16#8400;
      ErrProcessingIntern : Word := 16#8600;
      ErrAreaReserved : Word := 16#8800;
      ErrUserDefinedClasses : Word := 16#9000;
   END_VAR


BEGIN
	#txEnable := #xEnable;
	REGION ACTIVATION/DESACTIVATION
	  IF #txEnable AND #swStatus = #StatusNoCall THEN // Mise en service du bloc FB
	    #sxValid := FALSE;
	    #sxBusy := FALSE;
	    #sxError := FALSE;
	    #swStatus := #StatusFirstCall;
	    #sxErrorUserCleared := FALSE;
	    #sxErrorAutoCleared := FALSE;
	    #sxDisablingCompleted := FALSE;
	    #sdiFbState := #FB_StateEnabling;
	   
	  ELSIF ((NOT #txEnable) AND #sxEnabledOld) THEN // Desactivation du bloc FB
	    #sdiFbState := #FB_StateDisabling;
	    ;
	  ELSIF (#swStatus = #StatusFirstCall) THEN
	    #swStatus := #StatusSubsequenceCall;
	  END_IF;
	  
	  // Edge detection 'enable' input
	  #sxEnabledOld := #txEnable;
	END_REGION ACTIVATION/DESACTIVATION
	
	REGION APPEL BLOC FONCTION
	  #miDB_ModbusClient(REQ          := #sxMBcReq,
	                     DISCONNECT   := FALSE,
	                     MB_MODE      := 0,
	                     MB_DATA_ADDR := #sudiMBcAddress,
	                     MB_DATA_LEN  := #suiMBcLen,
	                     DONE         => #sxMBcDone,
	                     BUSY         => #sxMBcBusy,
	                     ERROR        => #sxMBcError,
	                     STATUS       => #swMBcStatus,
	                     MB_DATA_PTR  := #sarDataTemp,
	                     CONNECT      := #CommData);
	  
	  
	  #miDB_TonDelay(IN := #sxStartDelay,
	                 PT := #tDelay);
	  
	END_REGION APPEL BLOC FONCTION
	
	IF (#swStatus = #StatusNoCall) THEN // Nothing to do -> End here to reduce "system load"
	  RETURN;
	END_IF;
	
	REGION STATE MACHINE
	  CASE #sdiFbState OF
	      
	    #FB_StateNoProcessing:
	      REGION NoProcessing
	        #snStep := #StepInitial; // Step to init
	        #sxMBcReq := FALSE; // Raz request for MB client
	        #sxMBcDisconnect := TRUE; // Enable disconnecting
	        #sxStartDelay := FALSE; // Stop timer delay
	        IF #sxError AND #xReset THEN
	          #sxErrorUserCleared := FALSE;
	          ;//Do nothing more
	        END_IF;
	      END_REGION NoProcessing  
	      
	    #FB_StateEnabling:
	      REGION Enabling
	        #sxValid := FALSE;
	        #sxBusy := TRUE;
	        #sxError := FALSE;
	        #sxMBcDisconnect := FALSE;
	        #sxMBcReq := FALSE;
	        #sxStartDelay := FALSE;
	        #snStep := #StepInitial; //Initialisation du grafcet de fonctionnement
	        #sdiFbState := #FB_StateProcessing;
	      END_REGION Enabling
	      
	    #FB_StateProcessing:
	      REGION Processing
	        CASE #snStep OF
	            
	          #StepInitial:
	            #sudiMBcAddress := 40002;
	            #suiMBcLen := 70;
	            #snStep := #StepReqPhase1;
	            
	          #StepReqPhase1:
	            #sxMBcReq := TRUE;
	            IF #sxMBcBusy THEN
	              #snStep := #StepWaitDonePh1;
	            ELSIF #sxMBcError THEN
	              #sxMBcReq := FALSE;
	              #sxErrorUserCleared := TRUE;
	            END_IF;
	            
	          #StepWaitDonePh1:
	            IF #sxMBcDone THEN
	              #sxMBcReq := FALSE;
	              #snStep := #StepWriteDataPh1;
	            ELSIF #sxMBcError THEN
	              #sxMBcReq := FALSE;
	              #sxErrorUserCleared := TRUE;
	            END_IF;
	            
	          #StepWriteDataPh1:
	            #DataSentron.Voltage_PH_N_L1      := #sarDataTemp[0];
	            #DataSentron.Voltage_PH_N_L2      := #sarDataTemp[1];
	            #DataSentron.Voltage_PH_N_L3      := #sarDataTemp[2];
	            #DataSentron.Voltage_PH_PH_L12    := #sarDataTemp[3];
	            #DataSentron.Voltage_PH_PH_L23    := #sarDataTemp[4];
	            #DataSentron.Voltage_PH_PH_L31    := #sarDataTemp[5];
	            #DataSentron.Current_I_L1         := #sarDataTemp[6];
	            #DataSentron.Current_I_L2         := #sarDataTemp[7];
	            #DataSentron.Current_I_L3         := #sarDataTemp[8];
	            #DataSentron.Apparent_Power_L1    := #sarDataTemp[9] / 100.0;
	            #DataSentron.Apparent_Power_L2    := #sarDataTemp[10] / 100.0;
	            #DataSentron.Apparent_Power_L3 := #sarDataTemp[11] / 100.0;
	            #DataSentron.Active_Power_L1      := #sarDataTemp[12] / 100.0;
	            #DataSentron.Active_Power_L2      := #sarDataTemp[13] / 100.0;
	            #DataSentron.Active_Power_L3      := #sarDataTemp[14] / 100.0;
	            #DataSentron.Reactive_Power_L1    := #sarDataTemp[15] / 100.0;
	            #DataSentron.Reactive_Power_L2    := #sarDataTemp[16] / 100.0;
	            #DataSentron.Reactive_Power_L3    := #sarDataTemp[17] / 100.0;
	            #DataSentron.Power_Factor_L1      := #sarDataTemp[18] / 100.0;
	            #DataSentron.Power_Factor_L2      := #sarDataTemp[19] / 100.0;
	            #DataSentron.Power_Factor_L3      := #sarDataTemp[20] / 100.0;
	            #DataSentron.THD_R_V_L1           := #sarDataTemp[21];
	            #DataSentron.THD_R_V_L2           := #sarDataTemp[22];
	            #DataSentron.THD_R_V_L3           := #sarDataTemp[23];
	            #DataSentron.THD_R_I_L1           := #sarDataTemp[24];
	            #DataSentron.THD_R_I_L2           := #sarDataTemp[25];
	            #DataSentron.THD_R_I_L3           := #sarDataTemp[26];
	            #DataSentron.Frequency            := #sarDataTemp[27];
	            #DataSentron.Total_Apparent_Power := #sarDataTemp[31] / 100.0;
	            #DataSentron.Total_Active_Power   := #sarDataTemp[32] / 100.0;
	            #DataSentron.Total_Reactive_Power := #sarDataTemp[33] / 100.0;
	            #DataSentron.Total_Power_Factor   := #sarDataTemp[34] / 100.0;
	            #sudiMBcAddress := 40076;
	            #suiMBcLen := 70;
	            #snStep := #StepReqPhase2;
	            
	          #StepReqPhase2:
	            #sxMBcReq := TRUE;
	            IF #sxMBcBusy THEN
	              #snStep := #StepWaitDonePh2;
	            ELSIF #sxMBcError THEN
	              #sxMBcReq := FALSE;
	              #sxErrorUserCleared := TRUE;
	            END_IF;
	            
	          #StepWaitDonePh2:
	            IF #sxMBcDone THEN
	              #sxMBcReq := FALSE;
	              #snStep := #StepWriteDataPh2;
	            ELSIF #sxMBcError THEN
	              #sxMBcReq := FALSE;
	              #sxErrorUserCleared := TRUE;
	            END_IF;
	            
	          #StepWriteDataPh2:
	            #DataSentron.Voltage_PH_N_L1_MAX := #sarDataTemp[0];
	            #DataSentron.Voltage_PH_N_L2_MAX := #sarDataTemp[1];
	            #DataSentron.Voltage_PH_N_L3_MAX := #sarDataTemp[2];
	            #DataSentron.Voltage_PH_PH_L12_MAX := #sarDataTemp[3];
	            #DataSentron.Voltage_PH_PH_L23_MAX := #sarDataTemp[4];
	            #DataSentron.Voltage_PH_PH_L31_MAX := #sarDataTemp[5];
	            #DataSentron.Current_I_L1_MAX := #sarDataTemp[6];
	            #DataSentron.Current_I_L2_MAX := #sarDataTemp[7];
	            #DataSentron.Current_I_L3_MAX := #sarDataTemp[8];
	            #DataSentron.Apparent_Power_L1_MAX := #sarDataTemp[9] / 100.0;
	            #DataSentron.Apparent_Power_L2_MAX := #sarDataTemp[10] / 100.0;
	            #DataSentron.Apparent_Power_L3_MAX := #sarDataTemp[11] / 100.0;
	            #DataSentron.Active_Power_L1_MAX := #sarDataTemp[12] / 100.0;
	            #DataSentron.Active_Power_L2_MAX := #sarDataTemp[13] / 100.0;
	            #DataSentron.Active_Power_L3_MAX := #sarDataTemp[14] / 100.0;
	            #DataSentron.Reactive_Power_L1_MAX := #sarDataTemp[15] / 100.0;
	            #DataSentron.Reactive_Power_L2_MAX := #sarDataTemp[16] / 100.0;
	            #DataSentron.Reactive_Power_L3_MAX := #sarDataTemp[17] / 100.0;
	            #DataSentron.Power_Factor_L1_MAX := #sarDataTemp[18] / 100.0;
	            #DataSentron.Power_Factor_L2_MAX := #sarDataTemp[19] / 100.0;
	            #DataSentron.Power_Factor_L3_MAX := #sarDataTemp[20] / 100.0;
	            #DataSentron.THD_R_V_L1_MAX := #sarDataTemp[21];
	            #DataSentron.THD_R_V_L2_MAX := #sarDataTemp[22];
	            #DataSentron.THD_R_V_L3_MAX := #sarDataTemp[23];
	            #DataSentron.THD_R_I_L1_MAX := #sarDataTemp[24];
	            #DataSentron.THD_R_I_L2_MAX := #sarDataTemp[25];
	            #DataSentron.THD_R_I_L3_MAX := #sarDataTemp[26];
	            #DataSentron.Frequency_MAX := #sarDataTemp[27];
	            #DataSentron.Total_Apparent_Power_MAX := #sarDataTemp[31] / 100.0;
	            #DataSentron.Total_Active_Power_MAX := #sarDataTemp[32] / 100.0;
	            #DataSentron.Total_Reactive_Power_MAX := #sarDataTemp[33] / 100.0;
	            #DataSentron.Total_Power_Factor_MAX := #sarDataTemp[34] / 100.0;
	            #sudiMBcAddress := 40146;
	            #suiMBcLen := 58;
	            #snStep := #StepReqPhase3;
	            
	          #StepReqPhase3:
	            #sxMBcReq := TRUE;
	            IF #sxMBcBusy THEN
	              #snStep := #StepWaitDonePh3;
	            ELSIF #sxMBcError THEN
	              #sxMBcReq := FALSE;
	              #sxErrorUserCleared := TRUE;
	            END_IF;
	            
	          #StepWaitDonePh3:
	            IF #sxMBcDone THEN
	              #sxMBcReq := FALSE;
	              #snStep := #StepWriteDataPh3;
	            ELSIF #sxMBcError THEN
	              #sxMBcReq := FALSE;
	              #sxErrorUserCleared := TRUE;
	            END_IF;
	            
	          #StepWriteDataPh3:
	            #DataSentron.Voltage_PH_N_L1_MIN := #sarDataTemp[0];
	            #DataSentron.Voltage_PH_N_L2_MIN := #sarDataTemp[1];
	            #DataSentron.Voltage_PH_N_L3_MIN := #sarDataTemp[2];
	            #DataSentron.Voltage_PH_PH_L12_MIN := #sarDataTemp[3];
	            #DataSentron.Voltage_PH_PH_L23_MIN := #sarDataTemp[4];
	            #DataSentron.Voltage_PH_PH_L31_MIN := #sarDataTemp[5];
	            #DataSentron.Current_I_L1_MIN := #sarDataTemp[6];
	            #DataSentron.Current_I_L2_MIN := #sarDataTemp[7];
	            #DataSentron.Current_I_L3_MIN := #sarDataTemp[8];
	            #DataSentron.Apparent_Power_L1_MIN := #sarDataTemp[9] / 100.0;
	            #DataSentron.Apparent_Power_L2_MIN := #sarDataTemp[10] / 100.0;
	            #DataSentron.Apparent_Power_L3_MIN := #sarDataTemp[11] / 100.0;
	            #DataSentron.Active_Power_L1_MIN := #sarDataTemp[12] / 100.0;
	            #DataSentron.Active_Power_L2_MIN := #sarDataTemp[13] / 100.0;
	            #DataSentron.Active_Power_L3_MIN := #sarDataTemp[14] / 100.0;
	            #DataSentron.Reactive_Power_L1_MIN := #sarDataTemp[15] / 100.0;
	            #DataSentron.Reactive_Power_L2_MIN := #sarDataTemp[16] / 100.0;
	            #DataSentron.Reactive_Power_L3_MIN := #sarDataTemp[17] / 100.0;
	            #DataSentron.Power_Factor_L1_MIN := #sarDataTemp[18];
	            #DataSentron.Power_Factor_L2_MIN := #sarDataTemp[19];
	            #DataSentron.Power_Factor_L3_MIN := #sarDataTemp[20];
	            #DataSentron.Frequency_MIN := #sarDataTemp[21];
	            #DataSentron.Total_Apparent_Power_MIN := #sarDataTemp[25] / 100.0;
	            #DataSentron.Total_Active_Power_MIN := #sarDataTemp[26] / 100.0;
	            #DataSentron.Total_Reactive_Power_MIN := #sarDataTemp[27] / 100.0;
	            #DataSentron.Total_Power_Factor_MIN := #sarDataTemp[28] / 100.0;
	            #sudiMBcAddress := 0;
	            #suiMBcLen := 0;
	            #snStep := #StepWaitDelay;
	            
	          #StepWaitDelay:
	            #sxStartDelay := TRUE;
	            IF #miDB_TonDelay.Q THEN
	              #sxStartDelay := FALSE;
	              #snStep := #StepInitial;
	            END_IF;
	            
	          ELSE
	            // Si tu es la, t'as merdé un truc
	            ;
	        END_CASE;
	      END_REGION Processing
	      
	      
	    #FB_StateDisabling:
	      REGION Disabling 
	        #snStep := #StepInitial; //Initialisation du grafcet de fonctionnement
	        #sxMBcReq := FALSE;
	        #sxMBcDisconnect := TRUE;
	        #sxStartDelay := FALSE;
	        #sxDisablingCompleted := TRUE;
	        
	      END_REGION Disabling       
	    ELSE
	      REGION Undefined state
	        #swStatus := #ErrUndefinedState;
	        #sxErrorUserCleared := TRUE;
	      END_REGION Undefined sta      
	  END_CASE;
	  
	END_REGION STATE MACHINE
	    
	
	REGION SORTIES
	  IF #sxDisablingCompleted THEN
	    #sxValid := FALSE;
	    #sxBusy := FALSE;
	    #sxError := FALSE;
	    #sxErrorAutoCleared := FALSE;
	    #sxDisablingCompleted := FALSE;
	    #swStatus := #StatusNoCall;
	  ELSIF (#sxErrorUserCleared AND (NOT #sxError)) THEN
	    #sxValid := FALSE;
	    #sxBusy := FALSE;
	    #sxError := TRUE;
	    IF #sxMBcError THEN
	      #swStatus := #swMBcStatus;
	    END_IF;
	    #sdiFbState := #FB_StateNoProcessing;
	  ELSIF (#sxErrorAutoCleared AND  (NOT #sxError)) THEN
	    #sxValid := FALSE;
	    #sxBusy := TRUE;
	    #sxError := TRUE;
	  ELSIF ((NOT #sxErrorUserCleared) AND (NOT #sxErrorAutoCleared) AND #sxError) THEN
	    #sxValid := TRUE;
	    #sxBusy := TRUE;
	    #sxError := FALSE;
	    #sdiFbState := #FB_StateEnabling;
	    #swStatus := #StatusSubsequenceCall;
	  END_IF;
	END_REGION SORTIES
	
	REGION ECRITURE VALEURS DE SORTIES
	  #xValid := #sxValid;
	  #xBusy := #sxBusy;
	  #xError := #sxError;
	  #wStatus := #swStatus;
	  
	END_REGION ECRITURE VALEURS DE SORTIES
	
	
END_FUNCTION_BLOCK

FUNCTION "FC200_ServerNTP" : Void   // FC200, LAD
{ S7_Optimized_Access := 'TRUE' }
// stored: AutoNumber false, IsIECCheckEnabled true, SetENOAutomatically false
BEGIN

REGION Network 1: Server NTP (time)
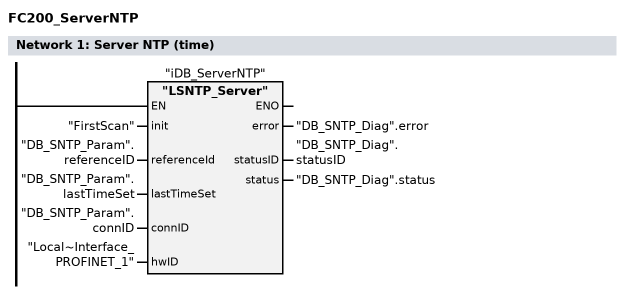
   RUNG wire#powerrail
      "iDB_ServerNTP"(init := "FirstScan", referenceId := "DB_SNTP_Param".referenceID, lastTimeSet := "DB_SNTP_Param".lastTimeSet, connID := "DB_SNTP_Param".connID, hwID := "Local~Interface_PROFINET_1", error => "DB_SNTP_Diag".error, statusID => "DB_SNTP_Diag".statusID, status => "DB_SNTP_Diag".status)
   END_RUNG
   // the same network as SCL:
   "iDB_ServerNTP"(init := "FirstScan",   // "LSNTP_Server"
                   referenceId := "DB_SNTP_Param".referenceID,
                   lastTimeSet := "DB_SNTP_Param".lastTimeSet,
                   connID := "DB_SNTP_Param".connID,
                   hwID := "Local~Interface_PROFINET_1",
                   error => "DB_SNTP_Diag".error,
                   statusID => "DB_SNTP_Diag".statusID,
                   status => "DB_SNTP_Diag".status);
END_REGION
END_FUNCTION

FUNCTION "FC900_SafetyIntegration" : Void   // FC900, F_LAD
{ S7_Optimized_Access := 'TRUE' }
// stored: AutoNumber false
BEGIN

REGION Network 1: Bit de reset
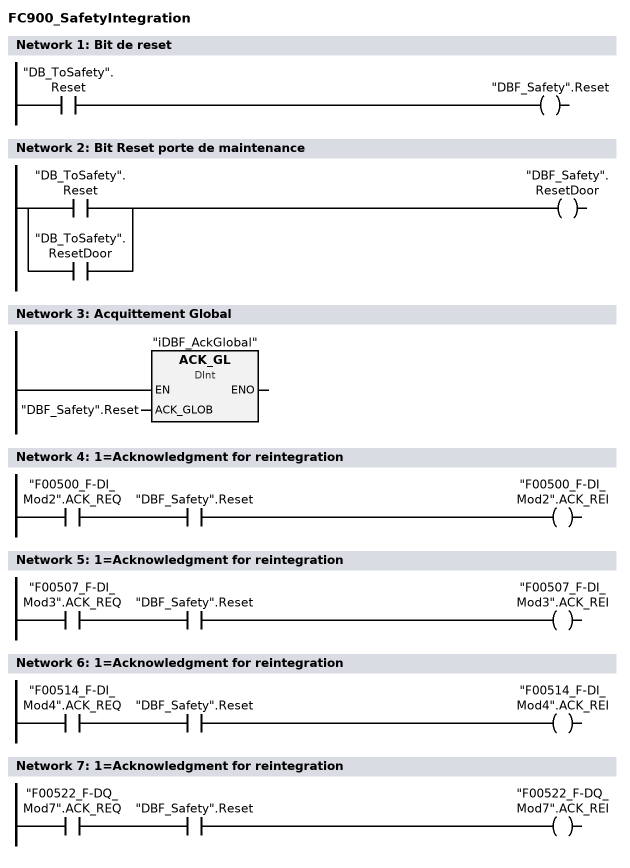
   RUNG wire#powerrail
      Contact( "DB_ToSafety".Reset )
      Coil( "DBF_Safety".Reset )
   END_RUNG
   // the same network as SCL:
   "DBF_Safety".Reset := "DB_ToSafety".Reset;
END_REGION

REGION Network 2: Bit Reset porte de maintenance
   RUNG wire#powerrail
      Contact( "DB_ToSafety".Reset )
      wire#w1
      Coil( "DBF_Safety".ResetDoor )
   END_RUNG
   RUNG wire#powerrail
      Contact( "DB_ToSafety".ResetDoor )
   END_RUNG wire#w1
   // the same network as SCL:
   "DBF_Safety".ResetDoor := "DB_ToSafety".Reset OR "DB_ToSafety".ResetDoor;
END_REGION

REGION Network 3: Acquittement Global
   RUNG wire#powerrail
      { S7_Templates := "codedbool_type := DInt" } "iDBF_AckGlobal".ACK_GL(ACK_GLOB := "DBF_Safety".Reset)
   END_RUNG
   // the same network as SCL:
   "iDBF_AckGlobal"(ACK_GLOB := "DBF_Safety".Reset);   // ACK_GL
END_REGION

REGION Network 4: 1=Acknowledgment for reintegration
   RUNG wire#powerrail
      Contact( "F00500_F-DI_Mod2".ACK_REQ )
      Contact( "DBF_Safety".Reset )
      Coil( "F00500_F-DI_Mod2".ACK_REI )
   END_RUNG
   // the same network as SCL:
   "F00500_F-DI_Mod2".ACK_REI := "F00500_F-DI_Mod2".ACK_REQ AND "DBF_Safety".Reset;
END_REGION

REGION Network 5: 1=Acknowledgment for reintegration
   RUNG wire#powerrail
      Contact( "F00507_F-DI_Mod3".ACK_REQ )
      Contact( "DBF_Safety".Reset )
      Coil( "F00507_F-DI_Mod3".ACK_REI )
   END_RUNG
   // the same network as SCL:
   "F00507_F-DI_Mod3".ACK_REI := "F00507_F-DI_Mod3".ACK_REQ AND "DBF_Safety".Reset;
END_REGION

REGION Network 6: 1=Acknowledgment for reintegration
   RUNG wire#powerrail
      Contact( "F00514_F-DI_Mod4".ACK_REQ )
      Contact( "DBF_Safety".Reset )
      Coil( "F00514_F-DI_Mod4".ACK_REI )
   END_RUNG
   // the same network as SCL:
   "F00514_F-DI_Mod4".ACK_REI := "F00514_F-DI_Mod4".ACK_REQ AND "DBF_Safety".Reset;
END_REGION

REGION Network 7: 1=Acknowledgment for reintegration
   RUNG wire#powerrail
      Contact( "F00522_F-DQ_Mod7".ACK_REQ )
      Contact( "DBF_Safety".Reset )
      Coil( "F00522_F-DQ_Mod7".ACK_REI )
   END_RUNG
   // the same network as SCL:
   "F00522_F-DQ_Mod7".ACK_REI := "F00522_F-DQ_Mod7".ACK_REQ AND "DBF_Safety".Reset;
END_REGION
END_FUNCTION

FUNCTION "FC901_SafetyInputs" : Void   // FC901, F_LAD
{ S7_Optimized_Access := 'TRUE' }
// stored: AutoNumber false
BEGIN

REGION Network 1: Emergency stop on main cabinet
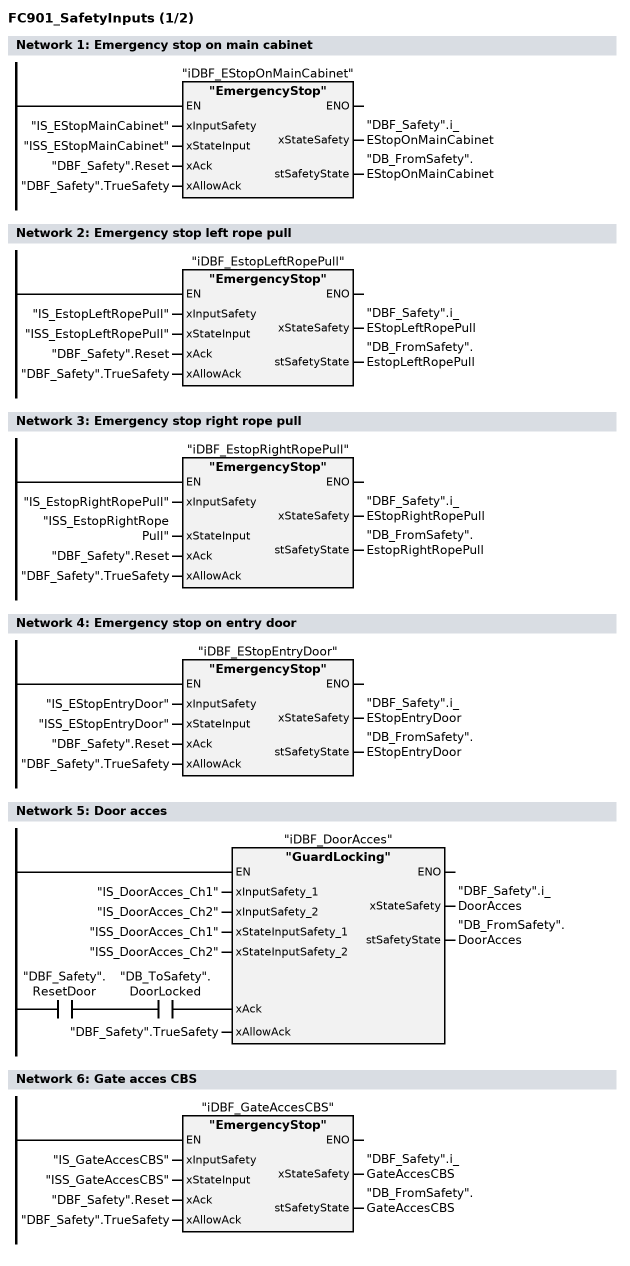
   RUNG wire#powerrail
      "iDBF_EStopOnMainCabinet"(xInputSafety := "IS_EStopMainCabinet", xStateInput := "ISS_EStopMainCabinet", xAck := "DBF_Safety".Reset, xAllowAck := "DBF_Safety".TrueSafety, xStateSafety => "DBF_Safety".i_EStopOnMainCabinet, stSafetyState => "DB_FromSafety".EStopOnMainCabinet)
   END_RUNG
   // the same network as SCL:
   "iDBF_EStopOnMainCabinet"(xInputSafety := "IS_EStopMainCabinet",   // "EmergencyStop"
                           xStateInput := "ISS_EStopMainCabinet",
                           xAck := "DBF_Safety".Reset,
                           xAllowAck := "DBF_Safety".TrueSafety,
                           xStateSafety => "DBF_Safety".i_EStopOnMainCabinet,
                           stSafetyState => "DB_FromSafety".EStopOnMainCabinet);
END_REGION

REGION Network 2: Emergency stop left rope pull
   RUNG wire#powerrail
      "iDBF_EstopLeftRopePull"(xInputSafety := "IS_EstopLeftRopePull", xStateInput := "ISS_EstopLeftRopePull", xAck := "DBF_Safety".Reset, xAllowAck := "DBF_Safety".TrueSafety, xStateSafety => "DBF_Safety".i_EStopLeftRopePull, stSafetyState => "DB_FromSafety".EstopLeftRopePull)
   END_RUNG
   // the same network as SCL:
   "iDBF_EstopLeftRopePull"(xInputSafety := "IS_EstopLeftRopePull",   // "EmergencyStop"
                           xStateInput := "ISS_EstopLeftRopePull",
                           xAck := "DBF_Safety".Reset,
                           xAllowAck := "DBF_Safety".TrueSafety,
                           xStateSafety => "DBF_Safety".i_EStopLeftRopePull,
                           stSafetyState => "DB_FromSafety".EstopLeftRopePull);
END_REGION

REGION Network 3: Emergency stop right rope pull
   RUNG wire#powerrail
      "iDBF_EstopRightRopePull"(xInputSafety := "IS_EstopRightRopePull", xStateInput := "ISS_EstopRightRopePull", xAck := "DBF_Safety".Reset, xAllowAck := "DBF_Safety".TrueSafety, xStateSafety => "DBF_Safety".i_EStopRightRopePull, stSafetyState => "DB_FromSafety".EstopRightRopePull)
   END_RUNG
   // the same network as SCL:
   "iDBF_EstopRightRopePull"(xInputSafety := "IS_EstopRightRopePull",   // "EmergencyStop"
                           xStateInput := "ISS_EstopRightRopePull",
                           xAck := "DBF_Safety".Reset,
                           xAllowAck := "DBF_Safety".TrueSafety,
                           xStateSafety => "DBF_Safety".i_EStopRightRopePull,
                           stSafetyState => "DB_FromSafety".EstopRightRopePull);
END_REGION

REGION Network 4: Emergency stop on entry door
   RUNG wire#powerrail
      "iDBF_EStopEntryDoor"(xInputSafety := "IS_EStopEntryDoor", xStateInput := "ISS_EStopEntryDoor", xAck := "DBF_Safety".Reset, xAllowAck := "DBF_Safety".TrueSafety, xStateSafety => "DBF_Safety".i_EStopEntryDoor, stSafetyState => "DB_FromSafety".EStopEntryDoor)
   END_RUNG
   // the same network as SCL:
   "iDBF_EStopEntryDoor"(xInputSafety := "IS_EStopEntryDoor",   // "EmergencyStop"
                         xStateInput := "ISS_EStopEntryDoor",
                         xAck := "DBF_Safety".Reset,
                         xAllowAck := "DBF_Safety".TrueSafety,
                         xStateSafety => "DBF_Safety".i_EStopEntryDoor,
                         stSafetyState => "DB_FromSafety".EStopEntryDoor);
END_REGION

REGION Network 5: Door acces
   RUNG wire#powerrail
      "iDBF_DoorAcces"(xAck := wire#w1, xInputSafety_1 := "IS_DoorAcces_Ch1", xInputSafety_2 := "IS_DoorAcces_Ch2", xStateInputSafety_1 := "ISS_DoorAcces_Ch1", xStateInputSafety_2 := "ISS_DoorAcces_Ch2", xAllowAck := "DBF_Safety".TrueSafety, xStateSafety => "DBF_Safety".i_DoorAcces, stSafetyState => "DB_FromSafety".DoorAcces)
   END_RUNG
   RUNG wire#powerrail
      Contact( "DBF_Safety".ResetDoor )
      Contact( "DB_ToSafety".DoorLocked )
   END_RUNG wire#w1
   // the same network as SCL:
   "iDBF_DoorAcces"(xInputSafety_1 := "IS_DoorAcces_Ch1",   // "GuardLocking"
                    xInputSafety_2 := "IS_DoorAcces_Ch2",
                    xStateInputSafety_1 := "ISS_DoorAcces_Ch1",
                    xStateInputSafety_2 := "ISS_DoorAcces_Ch2",
                    xAck := "DBF_Safety".ResetDoor AND "DB_ToSafety".DoorLocked,
                    xAllowAck := "DBF_Safety".TrueSafety,
                    xStateSafety => "DBF_Safety".i_DoorAcces,
                    stSafetyState => "DB_FromSafety".DoorAcces);
END_REGION

REGION Network 6: Gate acces CBS
   RUNG wire#powerrail
      "iDBF_GateAccesCBS"(xInputSafety := "IS_GateAccesCBS", xStateInput := "ISS_GateAccesCBS", xAck := "DBF_Safety".Reset, xAllowAck := "DBF_Safety".TrueSafety, xStateSafety => "DBF_Safety".i_GateAccesCBS, stSafetyState => "DB_FromSafety".GateAccesCBS)
   END_RUNG
   // the same network as SCL:
   "iDBF_GateAccesCBS"(xInputSafety := "IS_GateAccesCBS",   // "EmergencyStop"
                       xStateInput := "ISS_GateAccesCBS",
                       xAck := "DBF_Safety".Reset,
                       xAllowAck := "DBF_Safety".TrueSafety,
                       xStateSafety => "DBF_Safety".i_GateAccesCBS,
                       stSafetyState => "DB_FromSafety".GateAccesCBS);
END_REGION

REGION Network 7: Emergency stop in the control room
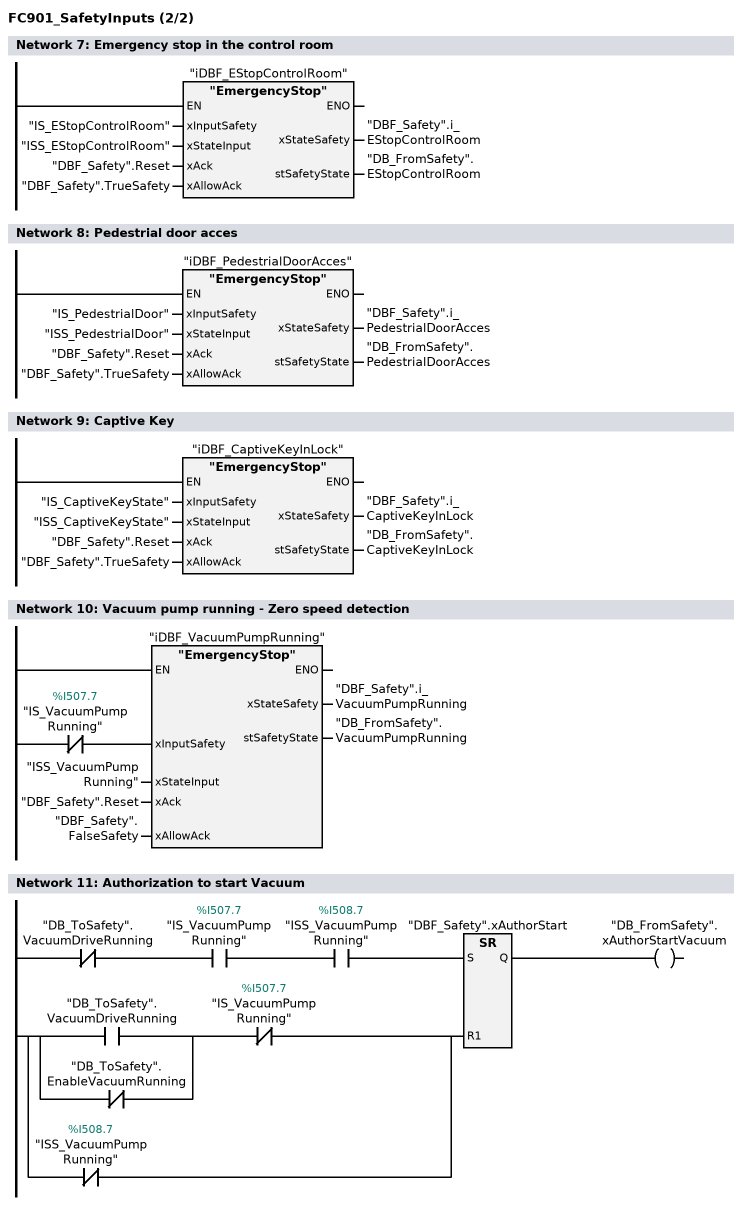
   RUNG wire#powerrail
      "iDBF_EStopControlRoom"(xInputSafety := "IS_EStopControlRoom", xStateInput := "ISS_EStopControlRoom", xAck := "DBF_Safety".Reset, xAllowAck := "DBF_Safety".TrueSafety, xStateSafety => "DBF_Safety".i_EStopControlRoom, stSafetyState => "DB_FromSafety".EStopControlRoom)
   END_RUNG
   // the same network as SCL:
   "iDBF_EStopControlRoom"(xInputSafety := "IS_EStopControlRoom",   // "EmergencyStop"
                           xStateInput := "ISS_EStopControlRoom",
                           xAck := "DBF_Safety".Reset,
                           xAllowAck := "DBF_Safety".TrueSafety,
                           xStateSafety => "DBF_Safety".i_EStopControlRoom,
                           stSafetyState => "DB_FromSafety".EStopControlRoom);
END_REGION

REGION Network 8: Pedestrial door acces
   RUNG wire#powerrail
      "iDBF_PedestrialDoorAcces"(xInputSafety := "IS_PedestrialDoor", xStateInput := "ISS_PedestrialDoor", xAck := "DBF_Safety".Reset, xAllowAck := "DBF_Safety".TrueSafety, xStateSafety => "DBF_Safety".i_PedestrialDoorAcces, stSafetyState => "DB_FromSafety".PedestrialDoorAcces)
   END_RUNG
   // the same network as SCL:
   "iDBF_PedestrialDoorAcces"(xInputSafety := "IS_PedestrialDoor",   // "EmergencyStop"
                           xStateInput := "ISS_PedestrialDoor",
                           xAck := "DBF_Safety".Reset,
                           xAllowAck := "DBF_Safety".TrueSafety,
                           xStateSafety => "DBF_Safety".i_PedestrialDoorAcces,
                           stSafetyState => "DB_FromSafety".PedestrialDoorAcces);
END_REGION

REGION Network 9: Captive Key
   RUNG wire#powerrail
      "iDBF_CaptiveKeyInLock"(xInputSafety := "IS_CaptiveKeyState", xStateInput := "ISS_CaptiveKeyState", xAck := "DBF_Safety".Reset, xAllowAck := "DBF_Safety".TrueSafety, xStateSafety => "DBF_Safety".i_CaptiveKeyInLock, stSafetyState => "DB_FromSafety".CaptiveKeyInLock)
   END_RUNG
   // the same network as SCL:
   "iDBF_CaptiveKeyInLock"(xInputSafety := "IS_CaptiveKeyState",   // "EmergencyStop"
                           xStateInput := "ISS_CaptiveKeyState",
                           xAck := "DBF_Safety".Reset,
                           xAllowAck := "DBF_Safety".TrueSafety,
                           xStateSafety => "DBF_Safety".i_CaptiveKeyInLock,
                           stSafetyState => "DB_FromSafety".CaptiveKeyInLock);
END_REGION

REGION Network 10: Vacuum pump running - Zero speed detection
   RUNG wire#powerrail
      "iDBF_VacuumPumpRunning"(xInputSafety := wire#w1, xStateInput := "ISS_VacuumPumpRunning", xAck := "DBF_Safety".Reset, xAllowAck := "DBF_Safety".FalseSafety, xStateSafety => "DBF_Safety".i_VacuumPumpRunning, stSafetyState => "DB_FromSafety".VacuumPumpRunning)
   END_RUNG
   RUNG wire#powerrail
      I_Contact( "IS_VacuumPumpRunning" )
   END_RUNG wire#w1
   // the same network as SCL:
   "iDBF_VacuumPumpRunning"(xInputSafety := NOT "IS_VacuumPumpRunning",   // "EmergencyStop"
                           xStateInput := "ISS_VacuumPumpRunning",
                           xAck := "DBF_Safety".Reset,
                           xAllowAck := "DBF_Safety".FalseSafety,
                           xStateSafety => "DBF_Safety".i_VacuumPumpRunning,
                           stSafetyState => "DB_FromSafety".VacuumPumpRunning);
END_REGION

REGION Network 11: Authorization to start Vacuum
   RUNG wire#powerrail
      I_Contact( "DB_ToSafety".VacuumDriveRunning )
      Contact( "IS_VacuumPumpRunning" )
      Contact( "ISS_VacuumPumpRunning" )
      S_SR(operand := "DBF_Safety".xAuthorStart, r1 := wire#w2)
      Coil( "DB_FromSafety".xAuthorStartVacuum )
   END_RUNG
   RUNG wire#powerrail
      Contact( "DB_ToSafety".VacuumDriveRunning )
      wire#w1
      I_Contact( "IS_VacuumPumpRunning" )
   END_RUNG wire#w2
   RUNG wire#powerrail
      I_Contact( "DB_ToSafety".EnableVacuumRunning )
   END_RUNG wire#w1
   RUNG wire#powerrail
      I_Contact( "ISS_VacuumPumpRunning" )
   END_RUNG wire#w2
   // the same network as SCL:
   IF NOT "DB_ToSafety".VacuumDriveRunning AND "IS_VacuumPumpRunning" AND "ISS_VacuumPumpRunning" THEN
       "DBF_Safety".xAuthorStart := TRUE;   // SR flip-flop
   END_IF;
   IF (("DB_ToSafety".VacuumDriveRunning OR NOT "DB_ToSafety".EnableVacuumRunning) AND NOT "IS_VacuumPumpRunning") OR NOT "ISS_VacuumPumpRunning" THEN
       "DBF_Safety".xAuthorStart := FALSE;
   END_IF;
   "DB_FromSafety".xAuthorStartVacuum := "DBF_Safety".xAuthorStart;
END_REGION
END_FUNCTION

FUNCTION "FC902_SafetyLogic" : Void   // FC902, F_LAD
{ S7_Optimized_Access := 'TRUE' }
// stored: AutoNumber false
BEGIN

REGION Network 1: Global Emergency Stop Cell
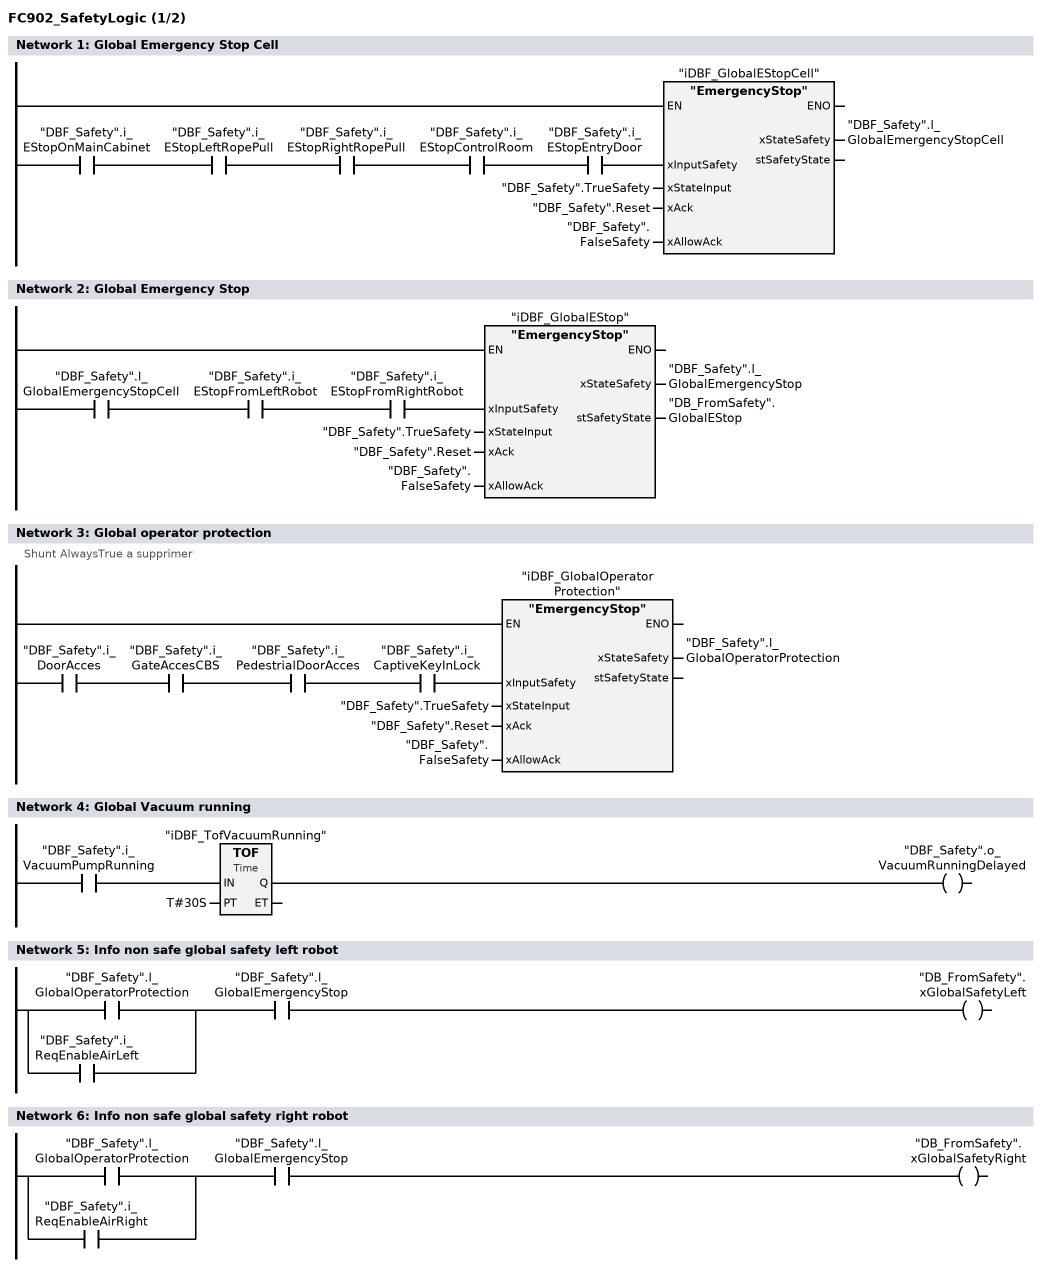
   RUNG wire#powerrail
      "iDBF_GlobalEStopCell"(xInputSafety := wire#w1, xStateInput := "DBF_Safety".TrueSafety, xAck := "DBF_Safety".Reset, xAllowAck := "DBF_Safety".FalseSafety, xStateSafety => "DBF_Safety".l_GlobalEmergencyStopCell, stSafetyState =>)
   END_RUNG
   RUNG wire#powerrail
      Contact( "DBF_Safety".i_EStopOnMainCabinet )
      Contact( "DBF_Safety".i_EStopLeftRopePull )
      Contact( "DBF_Safety".i_EStopRightRopePull )
      Contact( "DBF_Safety".i_EStopControlRoom )
      Contact( "DBF_Safety".i_EStopEntryDoor )
   END_RUNG wire#w1
   // the same network as SCL:
   "iDBF_GlobalEStopCell"(xInputSafety := "DBF_Safety".i_EStopOnMainCabinet AND "DBF_Safety".i_EStopLeftRopePull AND "DBF_Safety".i_EStopRightRopePull AND "DBF_Safety".i_EStopControlRoom AND "DBF_Safety".i_EStopEntryDoor,   // "EmergencyStop"
                          xStateInput := "DBF_Safety".TrueSafety,
                          xAck := "DBF_Safety".Reset,
                          xAllowAck := "DBF_Safety".FalseSafety,
                          xStateSafety => "DBF_Safety".l_GlobalEmergencyStopCell);
END_REGION

REGION Network 2: Global Emergency Stop
   RUNG wire#powerrail
      "iDBF_GlobalEStop"(xInputSafety := wire#w1, xStateInput := "DBF_Safety".TrueSafety, xAck := "DBF_Safety".Reset, xAllowAck := "DBF_Safety".FalseSafety, xStateSafety => "DBF_Safety".l_GlobalEmergencyStop, stSafetyState => "DB_FromSafety".GlobalEStop)
   END_RUNG
   RUNG wire#powerrail
      Contact( "DBF_Safety".l_GlobalEmergencyStopCell )
      Contact( "DBF_Safety".i_EStopFromLeftRobot )
      Contact( "DBF_Safety".i_EStopFromRightRobot )
   END_RUNG wire#w1
   // the same network as SCL:
   "iDBF_GlobalEStop"(xInputSafety := "DBF_Safety".l_GlobalEmergencyStopCell AND "DBF_Safety".i_EStopFromLeftRobot AND "DBF_Safety".i_EStopFromRightRobot,   // "EmergencyStop"
                      xStateInput := "DBF_Safety".TrueSafety,
                      xAck := "DBF_Safety".Reset,
                      xAllowAck := "DBF_Safety".FalseSafety,
                      xStateSafety => "DBF_Safety".l_GlobalEmergencyStop,
                      stSafetyState => "DB_FromSafety".GlobalEStop);
END_REGION

REGION Network 3: Global operator protection
   // Shunt AlwaysTrue a supprimer
   RUNG wire#powerrail
      "iDBF_GlobalOperatorProtection"(xInputSafety := wire#w1, xStateInput := "DBF_Safety".TrueSafety, xAck := "DBF_Safety".Reset, xAllowAck := "DBF_Safety".FalseSafety, xStateSafety => "DBF_Safety".l_GlobalOperatorProtection, stSafetyState =>)
   END_RUNG
   RUNG wire#powerrail
      Contact( "DBF_Safety".i_DoorAcces )
      Contact( "DBF_Safety".i_GateAccesCBS )
      Contact( "DBF_Safety".i_PedestrialDoorAcces )
      Contact( "DBF_Safety".i_CaptiveKeyInLock )
   END_RUNG wire#w1
   // the same network as SCL:
   "iDBF_GlobalOperatorProtection"(xInputSafety := "DBF_Safety".i_DoorAcces AND "DBF_Safety".i_GateAccesCBS AND "DBF_Safety".i_PedestrialDoorAcces AND "DBF_Safety".i_CaptiveKeyInLock,   // "EmergencyStop"
                           xStateInput := "DBF_Safety".TrueSafety,
                           xAck := "DBF_Safety".Reset,
                           xAllowAck := "DBF_Safety".FalseSafety,
                           xStateSafety => "DBF_Safety".l_GlobalOperatorProtection);
END_REGION

REGION Network 4: Global Vacuum running
   RUNG wire#powerrail
      Contact( "DBF_Safety".i_VacuumPumpRunning )
      { S7_Templates := "[time_type := Time, codedbool_type := DInt]" } "iDBF_TofVacuumRunning".TOF(pt := T#30S, et =>)
      Coil( "DBF_Safety".o_VacuumRunningDelayed )
   END_RUNG
   // the same network as SCL:
   "iDBF_TofVacuumRunning".TOF(IN := "DBF_Safety".i_VacuumPumpRunning, PT := T#30S);
   "DBF_Safety".o_VacuumRunningDelayed := "iDBF_TofVacuumRunning".Q;
END_REGION

REGION Network 5: Info non safe global safety left robot
   RUNG wire#powerrail
      Contact( "DBF_Safety".l_GlobalOperatorProtection )
      wire#w1
      Contact( "DBF_Safety".l_GlobalEmergencyStop )
      Coil( "DB_FromSafety".xGlobalSafetyLeft )
   END_RUNG
   RUNG wire#powerrail
      Contact( "DBF_Safety".i_ReqEnableAirLeft )
   END_RUNG wire#w1
   // the same network as SCL:
   "DB_FromSafety".xGlobalSafetyLeft := ("DBF_Safety".l_GlobalOperatorProtection OR "DBF_Safety".i_ReqEnableAirLeft) AND "DBF_Safety".l_GlobalEmergencyStop;
END_REGION

REGION Network 6: Info non safe global safety right robot
   RUNG wire#powerrail
      Contact( "DBF_Safety".l_GlobalOperatorProtection )
      wire#w1
      Contact( "DBF_Safety".l_GlobalEmergencyStop )
      Coil( "DB_FromSafety".xGlobalSafetyRight )
   END_RUNG
   RUNG wire#powerrail
      Contact( "DBF_Safety".i_ReqEnableAirRight )
   END_RUNG wire#w1
   // the same network as SCL:
   "DB_FromSafety".xGlobalSafetyRight := ("DBF_Safety".l_GlobalOperatorProtection OR "DBF_Safety".i_ReqEnableAirRight) AND "DBF_Safety".l_GlobalEmergencyStop;
END_REGION

REGION Network 7: Enable air pressure supply for left robot
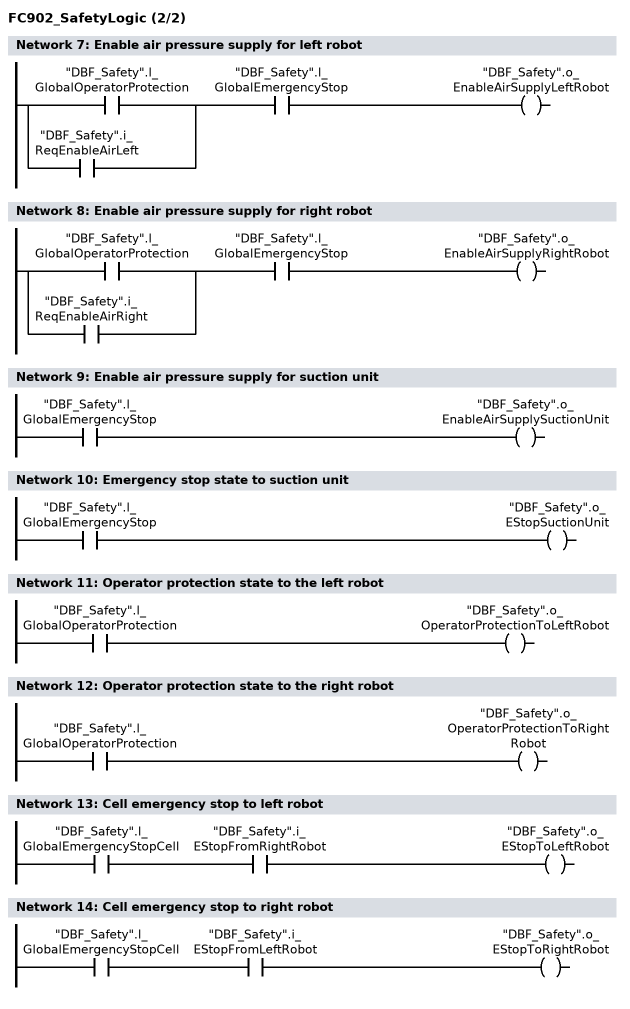
   RUNG wire#powerrail
      Contact( "DBF_Safety".l_GlobalOperatorProtection )
      wire#w1
      Contact( "DBF_Safety".l_GlobalEmergencyStop )
      Coil( "DBF_Safety".o_EnableAirSupplyLeftRobot )
   END_RUNG
   RUNG wire#powerrail
      Contact( "DBF_Safety".i_ReqEnableAirLeft )
   END_RUNG wire#w1
   // the same network as SCL:
   "DBF_Safety".o_EnableAirSupplyLeftRobot := ("DBF_Safety".l_GlobalOperatorProtection OR "DBF_Safety".i_ReqEnableAirLeft) AND "DBF_Safety".l_GlobalEmergencyStop;
END_REGION

REGION Network 8: Enable air pressure supply for right robot
   RUNG wire#powerrail
      Contact( "DBF_Safety".l_GlobalOperatorProtection )
      wire#w1
      Contact( "DBF_Safety".l_GlobalEmergencyStop )
      Coil( "DBF_Safety".o_EnableAirSupplyRightRobot )
   END_RUNG
   RUNG wire#powerrail
      Contact( "DBF_Safety".i_ReqEnableAirRight )
   END_RUNG wire#w1
   // the same network as SCL:
   "DBF_Safety".o_EnableAirSupplyRightRobot := ("DBF_Safety".l_GlobalOperatorProtection OR "DBF_Safety".i_ReqEnableAirRight) AND "DBF_Safety".l_GlobalEmergencyStop;
END_REGION

REGION Network 9: Enable air pressure supply for suction unit
   RUNG wire#powerrail
      Contact( "DBF_Safety".l_GlobalEmergencyStop )
      Coil( "DBF_Safety".o_EnableAirSupplySuctionUnit )
   END_RUNG
   // the same network as SCL:
   "DBF_Safety".o_EnableAirSupplySuctionUnit := "DBF_Safety".l_GlobalEmergencyStop;
END_REGION

REGION Network 10: Emergency stop state to suction unit
   RUNG wire#powerrail
      Contact( "DBF_Safety".l_GlobalEmergencyStop )
      Coil( "DBF_Safety".o_EStopSuctionUnit )
   END_RUNG
   // the same network as SCL:
   "DBF_Safety".o_EStopSuctionUnit := "DBF_Safety".l_GlobalEmergencyStop;
END_REGION

REGION Network 11: Operator protection state to the left robot
   RUNG wire#powerrail
      Contact( "DBF_Safety".l_GlobalOperatorProtection )
      Coil( "DBF_Safety".o_OperatorProtectionToLeftRobot )
   END_RUNG
   // the same network as SCL:
   "DBF_Safety".o_OperatorProtectionToLeftRobot := "DBF_Safety".l_GlobalOperatorProtection;
END_REGION

REGION Network 12: Operator protection state to the right robot
   RUNG wire#powerrail
      Contact( "DBF_Safety".l_GlobalOperatorProtection )
      Coil( "DBF_Safety".o_OperatorProtectionToRightRobot )
   END_RUNG
   // the same network as SCL:
   "DBF_Safety".o_OperatorProtectionToRightRobot := "DBF_Safety".l_GlobalOperatorProtection;
END_REGION

REGION Network 13: Cell emergency stop to left robot
   RUNG wire#powerrail
      Contact( "DBF_Safety".l_GlobalEmergencyStopCell )
      Contact( "DBF_Safety".i_EStopFromRightRobot )
      Coil( "DBF_Safety".o_EStopToLeftRobot )
   END_RUNG
   // the same network as SCL:
   "DBF_Safety".o_EStopToLeftRobot := "DBF_Safety".l_GlobalEmergencyStopCell AND "DBF_Safety".i_EStopFromRightRobot;
END_REGION

REGION Network 14: Cell emergency stop to right robot
   RUNG wire#powerrail
      Contact( "DBF_Safety".l_GlobalEmergencyStopCell )
      Contact( "DBF_Safety".i_EStopFromLeftRobot )
      Coil( "DBF_Safety".o_EStopToRightRobot )
   END_RUNG
   // the same network as SCL:
   "DBF_Safety".o_EStopToRightRobot := "DBF_Safety".l_GlobalEmergencyStopCell AND "DBF_Safety".i_EStopFromLeftRobot;
END_REGION
END_FUNCTION

FUNCTION "FC903_SafetyOutputs" : Void   // FC903, F_LAD
{ S7_Optimized_Access := 'TRUE' }
// stored: AutoNumber false
   VAR CONSTANT
      ct_FeedbackTime : Time := T#300ms;
   END_VAR
BEGIN

REGION Network 1: Enable air pressure supply on the left robot
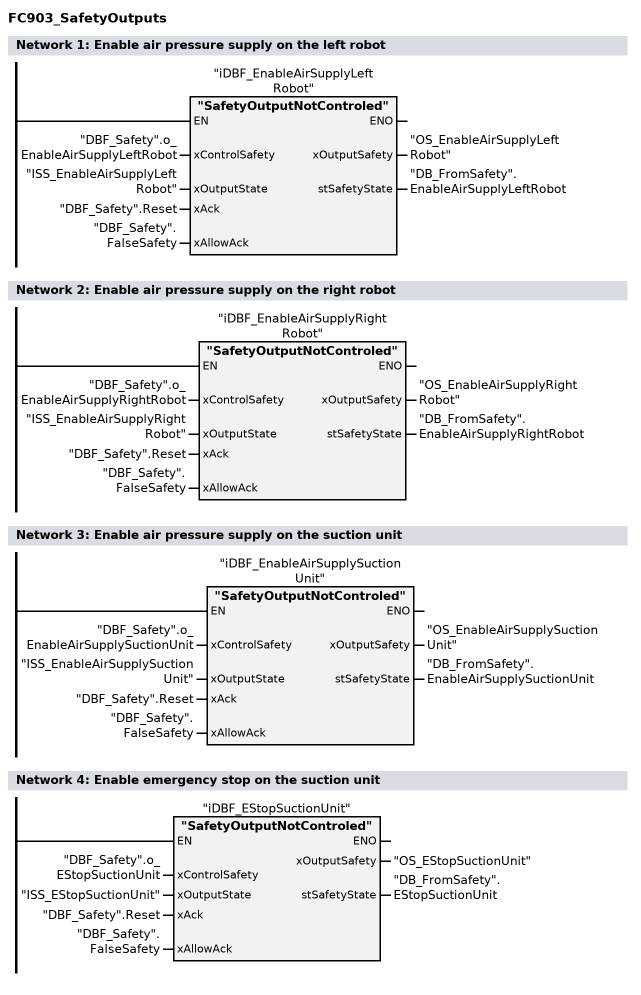
   RUNG wire#powerrail
      "iDBF_EnableAirSupplyLeftRobot"(xControlSafety := "DBF_Safety".o_EnableAirSupplyLeftRobot, xOutputState := "ISS_EnableAirSupplyLeftRobot", xAck := "DBF_Safety".Reset, xAllowAck := "DBF_Safety".FalseSafety, xOutputSafety => "OS_EnableAirSupplyLeftRobot", stSafetyState => "DB_FromSafety".EnableAirSupplyLeftRobot)
   END_RUNG
   // the same network as SCL:
   "iDBF_EnableAirSupplyLeftRobot"(xControlSafety := "DBF_Safety".o_EnableAirSupplyLeftRobot,   // "SafetyOutputNotControled"
                           xOutputState := "ISS_EnableAirSupplyLeftRobot",
                           xAck := "DBF_Safety".Reset,
                           xAllowAck := "DBF_Safety".FalseSafety,
                           xOutputSafety => "OS_EnableAirSupplyLeftRobot",
                           stSafetyState => "DB_FromSafety".EnableAirSupplyLeftRobot);
END_REGION

REGION Network 2: Enable air pressure supply on the right robot
   RUNG wire#powerrail
      "iDBF_EnableAirSupplyRightRobot"(xControlSafety := "DBF_Safety".o_EnableAirSupplyRightRobot, xOutputState := "ISS_EnableAirSupplyRightRobot", xAck := "DBF_Safety".Reset, xAllowAck := "DBF_Safety".FalseSafety, xOutputSafety => "OS_EnableAirSupplyRightRobot", stSafetyState => "DB_FromSafety".EnableAirSupplyRightRobot)
   END_RUNG
   // the same network as SCL:
   "iDBF_EnableAirSupplyRightRobot"(xControlSafety := "DBF_Safety".o_EnableAirSupplyRightRobot,   // "SafetyOutputNotControled"
                           xOutputState := "ISS_EnableAirSupplyRightRobot",
                           xAck := "DBF_Safety".Reset,
                           xAllowAck := "DBF_Safety".FalseSafety,
                           xOutputSafety => "OS_EnableAirSupplyRightRobot",
                           stSafetyState => "DB_FromSafety".EnableAirSupplyRightRobot);
END_REGION

REGION Network 3: Enable air pressure supply on the suction unit
   RUNG wire#powerrail
      "iDBF_EnableAirSupplySuctionUnit"(xControlSafety := "DBF_Safety".o_EnableAirSupplySuctionUnit, xOutputState := "ISS_EnableAirSupplySuctionUnit", xAck := "DBF_Safety".Reset, xAllowAck := "DBF_Safety".FalseSafety, xOutputSafety => "OS_EnableAirSupplySuctionUnit", stSafetyState => "DB_FromSafety".EnableAirSupplySuctionUnit)
   END_RUNG
   // the same network as SCL:
   "iDBF_EnableAirSupplySuctionUnit"(xControlSafety := "DBF_Safety".o_EnableAirSupplySuctionUnit,   // "SafetyOutputNotControled"
                           xOutputState := "ISS_EnableAirSupplySuctionUnit",
                           xAck := "DBF_Safety".Reset,
                           xAllowAck := "DBF_Safety".FalseSafety,
                           xOutputSafety => "OS_EnableAirSupplySuctionUnit",
                           stSafetyState => "DB_FromSafety".EnableAirSupplySuctionUnit);
END_REGION

REGION Network 4: Enable emergency stop on the suction unit
   RUNG wire#powerrail
      "iDBF_EStopSuctionUnit"(xControlSafety := "DBF_Safety".o_EStopSuctionUnit, xOutputState := "ISS_EStopSuctionUnit", xAck := "DBF_Safety".Reset, xAllowAck := "DBF_Safety".FalseSafety, xOutputSafety => "OS_EStopSuctionUnit", stSafetyState => "DB_FromSafety".EStopSuctionUnit)
   END_RUNG
   // the same network as SCL:
   "iDBF_EStopSuctionUnit"(xControlSafety := "DBF_Safety".o_EStopSuctionUnit,   // "SafetyOutputNotControled"
                           xOutputState := "ISS_EStopSuctionUnit",
                           xAck := "DBF_Safety".Reset,
                           xAllowAck := "DBF_Safety".FalseSafety,
                           xOutputSafety => "OS_EStopSuctionUnit",
                           stSafetyState => "DB_FromSafety".EStopSuctionUnit);
END_REGION
END_FUNCTION

FUNCTION_BLOCK "MainSafety"   // FB900, F_LAD
{ S7_Optimized_Access := 'TRUE' }
// stored: AutoNumber false
BEGIN

REGION Network 1: Read input safety from left robot
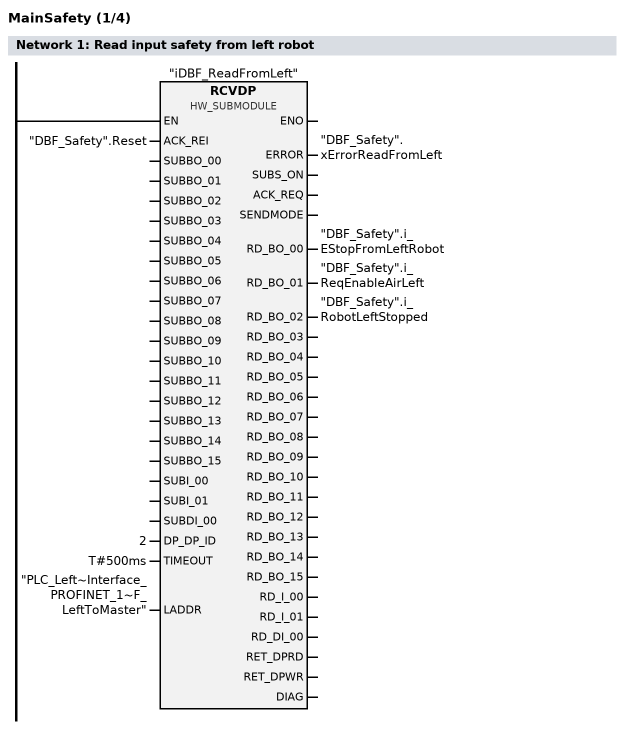
   RUNG wire#powerrail
      { S7_Templates := "laddr_type := HW_SUBMODULE" } "iDBF_ReadFromLeft".RCVDP(ACK_REI := "DBF_Safety".Reset, SUBBO_00 :=, SUBBO_01 :=, SUBBO_02 :=, SUBBO_03 :=, SUBBO_04 :=, SUBBO_05 :=, SUBBO_06 :=, SUBBO_07 :=, SUBBO_08 :=, SUBBO_09 :=, SUBBO_10 :=, SUBBO_11 :=, SUBBO_12 :=, SUBBO_13 :=, SUBBO_14 :=, SUBBO_15 :=, SUBI_00 :=, SUBI_01 :=, SUBDI_00 :=, DP_DP_ID := 2, TIMEOUT := T#500ms, LADDR := "PLC_Left~Interface_PROFINET_1~F_LeftToMaster", ERROR => "DBF_Safety".xErrorReadFromLeft, SUBS_ON =>, ACK_REQ =>, SENDMODE =>, RD_BO_00 => "DBF_Safety".i_EStopFromLeftRobot, RD_BO_01 => "DBF_Safety".i_ReqEnableAirLeft, RD_BO_02 => "DBF_Safety".i_RobotLeftStopped, RD_BO_03 =>, RD_BO_04 =>, RD_BO_05 =>, RD_BO_06 =>, RD_BO_07 =>, RD_BO_08 =>, RD_BO_09 =>, RD_BO_10 =>, RD_BO_11 =>, RD_BO_12 =>, RD_BO_13 =>, RD_BO_14 =>, RD_BO_15 =>, RD_I_00 =>, RD_I_01 =>, RD_DI_00 =>, RET_DPRD =>, RET_DPWR =>, DIAG =>)
   END_RUNG
   // the same network as SCL:
   "iDBF_ReadFromLeft"(ACK_REI := "DBF_Safety".Reset,   // RCVDP
                       DP_DP_ID := 2,
                       TIMEOUT := T#500ms,
                       LADDR := "PLC_Left~Interface_PROFINET_1~F_LeftToMaster",
                       ERROR => "DBF_Safety".xErrorReadFromLeft,
                       RD_BO_00 => "DBF_Safety".i_EStopFromLeftRobot,
                       RD_BO_01 => "DBF_Safety".i_ReqEnableAirLeft,
                       RD_BO_02 => "DBF_Safety".i_RobotLeftStopped);
END_REGION

REGION Network 2: Read input safety from right robot
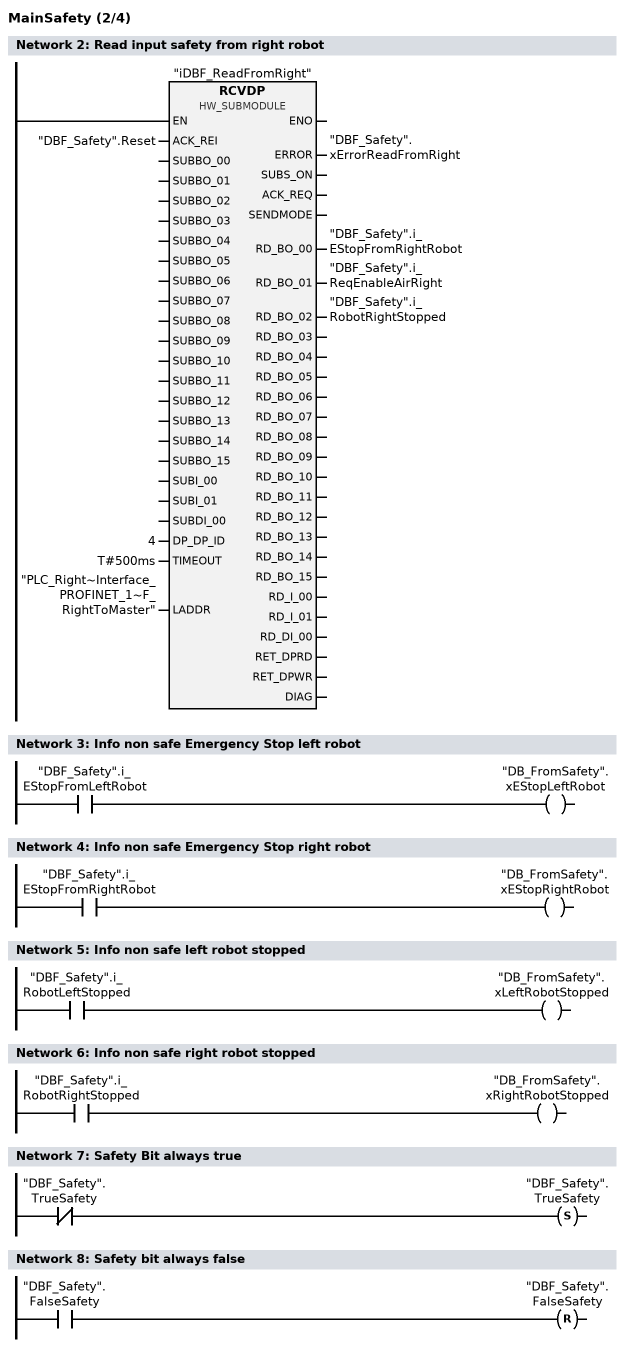
   RUNG wire#powerrail
      { S7_Templates := "laddr_type := HW_SUBMODULE" } "iDBF_ReadFromRight".RCVDP(ACK_REI := "DBF_Safety".Reset, SUBBO_00 :=, SUBBO_01 :=, SUBBO_02 :=, SUBBO_03 :=, SUBBO_04 :=, SUBBO_05 :=, SUBBO_06 :=, SUBBO_07 :=, SUBBO_08 :=, SUBBO_09 :=, SUBBO_10 :=, SUBBO_11 :=, SUBBO_12 :=, SUBBO_13 :=, SUBBO_14 :=, SUBBO_15 :=, SUBI_00 :=, SUBI_01 :=, SUBDI_00 :=, DP_DP_ID := 4, TIMEOUT := T#500ms, LADDR := "PLC_Right~Interface_PROFINET_1~F_RightToMaster", ERROR => "DBF_Safety".xErrorReadFromRight, SUBS_ON =>, ACK_REQ =>, SENDMODE =>, RD_BO_00 => "DBF_Safety".i_EStopFromRightRobot, RD_BO_01 => "DBF_Safety".i_ReqEnableAirRight, RD_BO_02 => "DBF_Safety".i_RobotRightStopped, RD_BO_03 =>, RD_BO_04 =>, RD_BO_05 =>, RD_BO_06 =>, RD_BO_07 =>, RD_BO_08 =>, RD_BO_09 =>, RD_BO_10 =>, RD_BO_11 =>, RD_BO_12 =>, RD_BO_13 =>, RD_BO_14 =>, RD_BO_15 =>, RD_I_00 =>, RD_I_01 =>, RD_DI_00 =>, RET_DPRD =>, RET_DPWR =>, DIAG =>)
   END_RUNG
   // the same network as SCL:
   "iDBF_ReadFromRight"(ACK_REI := "DBF_Safety".Reset,   // RCVDP
                        DP_DP_ID := 4,
                        TIMEOUT := T#500ms,
                        LADDR := "PLC_Right~Interface_PROFINET_1~F_RightToMaster",
                        ERROR => "DBF_Safety".xErrorReadFromRight,
                        RD_BO_00 => "DBF_Safety".i_EStopFromRightRobot,
                        RD_BO_01 => "DBF_Safety".i_ReqEnableAirRight,
                        RD_BO_02 => "DBF_Safety".i_RobotRightStopped);
END_REGION

REGION Network 3: Info non safe Emergency Stop left robot
   RUNG wire#powerrail
      Contact( "DBF_Safety".i_EStopFromLeftRobot )
      Coil( "DB_FromSafety".xEStopLeftRobot )
   END_RUNG
   // the same network as SCL:
   "DB_FromSafety".xEStopLeftRobot := "DBF_Safety".i_EStopFromLeftRobot;
END_REGION

REGION Network 4: Info non safe Emergency Stop right robot
   RUNG wire#powerrail
      Contact( "DBF_Safety".i_EStopFromRightRobot )
      Coil( "DB_FromSafety".xEStopRightRobot )
   END_RUNG
   // the same network as SCL:
   "DB_FromSafety".xEStopRightRobot := "DBF_Safety".i_EStopFromRightRobot;
END_REGION

REGION Network 5: Info non safe left robot stopped
   RUNG wire#powerrail
      Contact( "DBF_Safety".i_RobotLeftStopped )
      Coil( "DB_FromSafety".xLeftRobotStopped )
   END_RUNG
   // the same network as SCL:
   "DB_FromSafety".xLeftRobotStopped := "DBF_Safety".i_RobotLeftStopped;
END_REGION

REGION Network 6: Info non safe right robot stopped
   RUNG wire#powerrail
      Contact( "DBF_Safety".i_RobotRightStopped )
      Coil( "DB_FromSafety".xRightRobotStopped )
   END_RUNG
   // the same network as SCL:
   "DB_FromSafety".xRightRobotStopped := "DBF_Safety".i_RobotRightStopped;
END_REGION

REGION Network 7: Safety Bit always true
   RUNG wire#powerrail
      I_Contact( "DBF_Safety".TrueSafety )
      S_Coil( "DBF_Safety".TrueSafety )
   END_RUNG
   // the same network as SCL:
   IF NOT "DBF_Safety".TrueSafety THEN "DBF_Safety".TrueSafety := TRUE; END_IF;
END_REGION

REGION Network 8: Safety bit always false
   RUNG wire#powerrail
      Contact( "DBF_Safety".FalseSafety )
      R_Coil( "DBF_Safety".FalseSafety )
   END_RUNG
   // the same network as SCL:
   IF "DBF_Safety".FalseSafety THEN "DBF_Safety".FalseSafety := FALSE; END_IF;
END_REGION

REGION Network 9: Safety reintegration function call
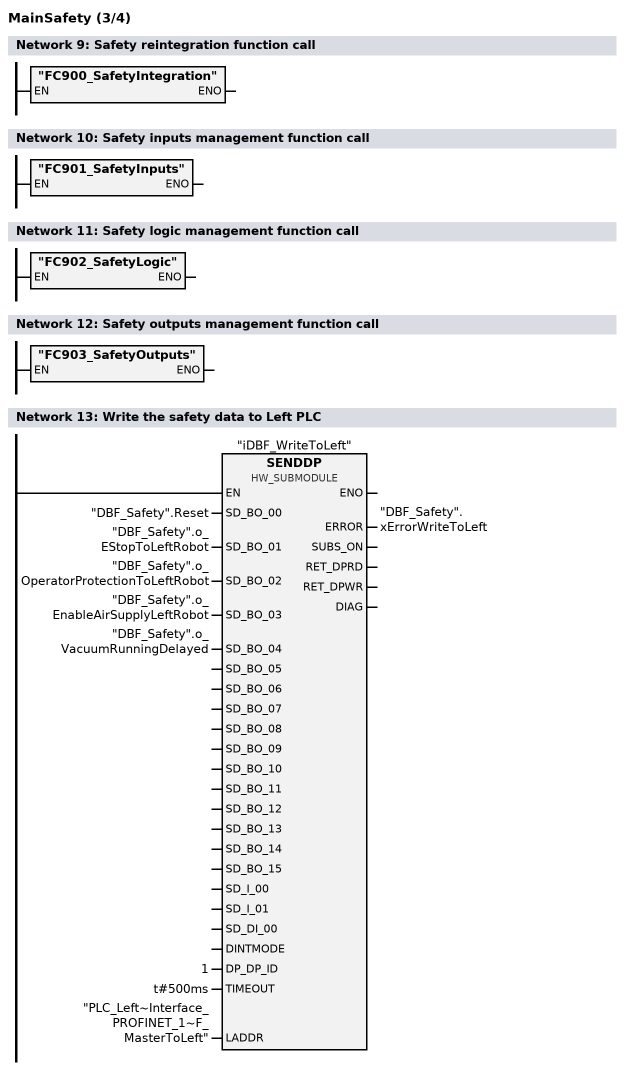
   RUNG wire#powerrail
      "FC900_SafetyIntegration"()
   END_RUNG
   // the same network as SCL:
   "FC900_SafetyIntegration"();
END_REGION

REGION Network 10: Safety inputs management function call
   RUNG wire#powerrail
      "FC901_SafetyInputs"()
   END_RUNG
   // the same network as SCL:
   "FC901_SafetyInputs"();
END_REGION

REGION Network 11: Safety logic management function call
   RUNG wire#powerrail
      "FC902_SafetyLogic"()
   END_RUNG
   // the same network as SCL:
   "FC902_SafetyLogic"();
END_REGION

REGION Network 12: Safety outputs management function call
   RUNG wire#powerrail
      "FC903_SafetyOutputs"()
   END_RUNG
   // the same network as SCL:
   "FC903_SafetyOutputs"();
END_REGION

REGION Network 13: Write the safety data to Left PLC
   RUNG wire#powerrail
      { S7_Templates := "laddr_type := HW_SUBMODULE" } "iDBF_WriteToLeft".SENDDP(SD_BO_00 := "DBF_Safety".Reset, SD_BO_01 := "DBF_Safety".o_EStopToLeftRobot, SD_BO_02 := "DBF_Safety".o_OperatorProtectionToLeftRobot, SD_BO_03 := "DBF_Safety".o_EnableAirSupplyLeftRobot, SD_BO_04 := "DBF_Safety".o_VacuumRunningDelayed, SD_BO_05 :=, SD_BO_06 :=, SD_BO_07 :=, SD_BO_08 :=, SD_BO_09 :=, SD_BO_10 :=, SD_BO_11 :=, SD_BO_12 :=, SD_BO_13 :=, SD_BO_14 :=, SD_BO_15 :=, SD_I_00 :=, SD_I_01 :=, SD_DI_00 :=, DINTMODE :=, DP_DP_ID := 1, TIMEOUT := t#500ms, LADDR := "PLC_Left~Interface_PROFINET_1~F_MasterToLeft", ERROR => "DBF_Safety".xErrorWriteToLeft, SUBS_ON =>, RET_DPRD =>, RET_DPWR =>, DIAG =>)
   END_RUNG
   // the same network as SCL:
   "iDBF_WriteToLeft"(SD_BO_00 := "DBF_Safety".Reset,   // SENDDP
                      SD_BO_01 := "DBF_Safety".o_EStopToLeftRobot,
                      SD_BO_02 := "DBF_Safety".o_OperatorProtectionToLeftRobot,
                      SD_BO_03 := "DBF_Safety".o_EnableAirSupplyLeftRobot,
                      SD_BO_04 := "DBF_Safety".o_VacuumRunningDelayed,
                      DP_DP_ID := 1,
                      TIMEOUT := t#500ms,
                      LADDR := "PLC_Left~Interface_PROFINET_1~F_MasterToLeft",
                      ERROR => "DBF_Safety".xErrorWriteToLeft);
END_REGION

REGION Network 14: Write the safety data to Right PLC
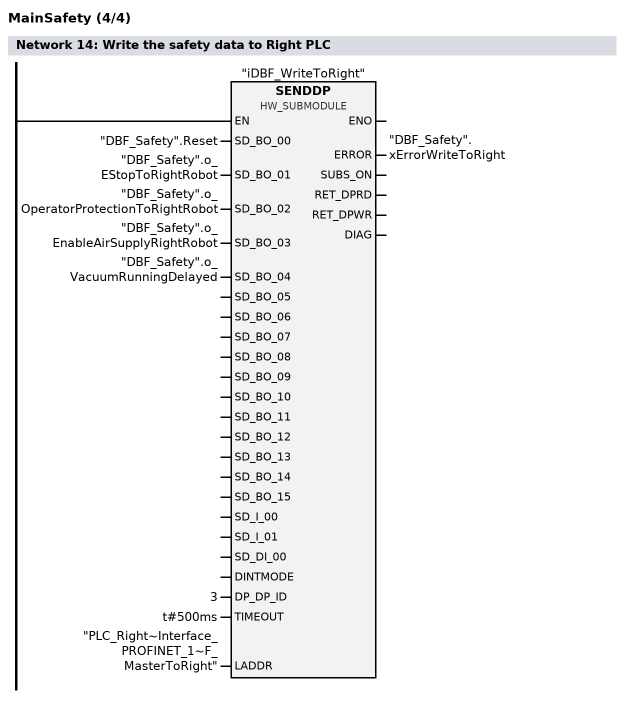
   RUNG wire#powerrail
      { S7_Templates := "laddr_type := HW_SUBMODULE" } "iDBF_WriteToRight".SENDDP(SD_BO_00 := "DBF_Safety".Reset, SD_BO_01 := "DBF_Safety".o_EStopToRightRobot, SD_BO_02 := "DBF_Safety".o_OperatorProtectionToRightRobot, SD_BO_03 := "DBF_Safety".o_EnableAirSupplyRightRobot, SD_BO_04 := "DBF_Safety".o_VacuumRunningDelayed, SD_BO_05 :=, SD_BO_06 :=, SD_BO_07 :=, SD_BO_08 :=, SD_BO_09 :=, SD_BO_10 :=, SD_BO_11 :=, SD_BO_12 :=, SD_BO_13 :=, SD_BO_14 :=, SD_BO_15 :=, SD_I_00 :=, SD_I_01 :=, SD_DI_00 :=, DINTMODE :=, DP_DP_ID := 3, TIMEOUT := t#500ms, LADDR := "PLC_Right~Interface_PROFINET_1~F_MasterToRight", ERROR => "DBF_Safety".xErrorWriteToRight, SUBS_ON =>, RET_DPRD =>, RET_DPWR =>, DIAG =>)
   END_RUNG
   // the same network as SCL:
   "iDBF_WriteToRight"(SD_BO_00 := "DBF_Safety".Reset,   // SENDDP
                       SD_BO_01 := "DBF_Safety".o_EStopToRightRobot,
                       SD_BO_02 := "DBF_Safety".o_OperatorProtectionToRightRobot,
                       SD_BO_03 := "DBF_Safety".o_EnableAirSupplyRightRobot,
                       SD_BO_04 := "DBF_Safety".o_VacuumRunningDelayed,
                       DP_DP_ID := 3,
                       TIMEOUT := t#500ms,
                       LADDR := "PLC_Right~Interface_PROFINET_1~F_MasterToRight",
                       ERROR => "DBF_Safety".xErrorWriteToRight);
END_REGION
END_FUNCTION_BLOCK

FUNCTION_BLOCK "FB22_DisplayRecipe"
{ S7_Optimized_Access := 'TRUE' }
VERSION : 0.1
   VAR_INPUT 
      xRecipeOpeInProgress { ExternalAccessible := 'False'; ExternalVisible := 'False'; ExternalWritable := 'False'} : Bool;   // Recipe operantion in progress
      xSaveRecipe { ExternalAccessible := 'False'; ExternalVisible := 'False'; ExternalWritable := 'False'} : Bool;   // Save current recipe into the data base
      xNextRecipe { ExternalAccessible := 'False'; ExternalVisible := 'False'; ExternalWritable := 'False'} : Bool;   // Load next recipe in the data base
      xPrevRecipe { ExternalAccessible := 'False'; ExternalVisible := 'False'; ExternalWritable := 'False'} : Bool;   // Load previus recipe in the data base
   END_VAR


BEGIN
END_FUNCTION_BLOCK

DATA_BLOCK "iDB_ManageVacuum"   // DB10
{ DB_Accessible_From_OPC_UA := 'FALSE' }
// stored: AutoNumber false, DBAccessibleFromOPCUA false, DBAccessibleFromWebserver false, InstanceOfName FB10_ManageVacuum, InstanceOfType FB
"FB10_ManageVacuum"
BEGIN
END_DATA_BLOCK

DATA_BLOCK "iDB_RunningTime"   // DB11
// stored: AutoNumber false, InstanceOfName FB_TimeCounter, InstanceOfType FB
"FB_TimeCounter"
   // VAR_INPUT
   //    xClockSecond { ExternalAccessible := 'False'; ExternalVisible := 'False'; ExternalWritable := 'False'} : Bool;
   //    xStart { ExternalAccessible := 'False'; ExternalVisible := 'False'; ExternalWritable := 'False'} : Bool;
   //    xStop { ExternalAccessible := 'False'; ExternalVisible := 'False'; ExternalWritable := 'False'} : Bool;
   //    xResetCounter { ExternalAccessible := 'False'; ExternalVisible := 'False'; ExternalWritable := 'False'} : Bool;
   // END_VAR
   // VAR_OUTPUT
   //    PerpetualCounter { ExternalAccessible := 'False'; ExternalVisible := 'False'; ExternalWritable := 'False'} : UDInt;
   //    "Counter" { ExternalAccessible := 'False'; ExternalVisible := 'False'; ExternalWritable := 'False'} : UDInt;
   // END_VAR
   // VAR
   //    sxEnableCount { ExternalAccessible := 'False'; ExternalVisible := 'False'; ExternalWritable := 'False'} : Bool;
   //    sxFpStart { ExternalAccessible := 'False'; ExternalVisible := 'False'; ExternalWritable := 'False'} : Bool;
   //    sxFpStop { ExternalAccessible := 'False'; ExternalVisible := 'False'; ExternalWritable := 'False'} : Bool;
   // END_VAR
   // VAR RETAIN
   //    miDB_Counter { ExternalAccessible := 'False'; ExternalVisible := 'False'; ExternalWritable := 'False'; S7_SetPoint := 'True'} : CTU_UDINT;
   //    miDB_PerpetualCount { ExternalAccessible := 'False'; ExternalVisible := 'False'; ExternalWritable := 'False'; S7_SetPoint := 'True'} : CTU_UDINT;
   // END_VAR
   // VAR
   //    sxFpResetCounter { ExternalAccessible := 'False'; ExternalVisible := 'False'; ExternalWritable := 'False'} : Bool;
   //    sxResetCounter { ExternalAccessible := 'False'; ExternalVisible := 'False'; ExternalWritable := 'False'} : Bool;
   // END_VAR
BEGIN
END_DATA_BLOCK

DATA_BLOCK "iDB_ManageState"   // DB20
{ DB_Accessible_From_OPC_UA := 'FALSE' }
// stored: AutoNumber false, DBAccessibleFromOPCUA false, DBAccessibleFromWebserver false, InstanceOfName FB20_ManageState, InstanceOfType FB
"FB20_ManageState"
BEGIN
END_DATA_BLOCK

DATA_BLOCK "iDB_ManageTowerLight"   // DB21
{ DB_Accessible_From_OPC_UA := 'FALSE' }
// stored: AutoNumber false, DBAccessibleFromOPCUA false, DBAccessibleFromWebserver false, InstanceOfName FB21_ManageTowerLight, InstanceOfType FB
"FB21_ManageTowerLight"
BEGIN
END_DATA_BLOCK

DATA_BLOCK "iDB_ServerNTP"   // DB200
{ DB_Accessible_From_OPC_UA := 'FALSE' }
VERSION : 2.1
// stored: AutoNumber false, DBAccessibleFromOPCUA false, DBAccessibleFromWebserver false, InstanceOfName LSNTP_Server, InstanceOfType FB
"LSNTP_Server"
   // VAR_INPUT
   //    init : Bool;
   //    referenceId : USInt;
   //    lastTimeSet : DTL;
   //    connID : CONN_OUC;
   //    hwID : HW_ANY;
   // END_VAR
   // VAR_OUTPUT
   //    error : Bool;
   //    statusID : Int;
   //    status : Word;
   // END_VAR
   // VAR
   //    InstTCON { S7_SetPoint := 'True'} : TCON;
   //    InstTURCV { S7_SetPoint := 'True'} : TURCV;
   //    InstTUSEND { S7_SetPoint := 'True'} : TUSEND;
   //    InstTDISCON { S7_SetPoint := 'True'} : TDISCON;
   //    statDiscon : Struct
   //       req : Bool;
   //       done : Bool;
   //       error : Bool;
   //       status : Word;
   //    END_STRUCT;
   //    statCon : Struct
   //       req : Bool;
   //       done : Bool;
   //       error : Bool;
   //       status : Word;
   //       param { S7_SetPoint := 'True'} : TCON_IP_v4;
   //    END_STRUCT;
   //    statRcv : Struct
   //       req : Bool;
   //       busy : Bool;
   //       error : Bool;
   //       ndr : Bool;
   //       len : UDInt;
   //       status : Word;
   //       addr { S7_SetPoint := 'True'} : TADDR_Param;
   //       tel { S7_SetPoint := 'True'} : "LSNTP_typeTelegram";
   //    END_STRUCT;
   //    statSend : Struct
   //       req : Bool;
   //       done : Bool;
   //       reqDone : Bool;
   //       error : Bool;
   //       status : Word;
   //       addr { S7_SetPoint := 'True'} : TADDR_Param;
   //       tel { S7_SetPoint := 'True'} : "LSNTP_typeTelegram";
   //    END_STRUCT;
   //    statState : Int;
   //    statEdge : Struct
   //       init : Bool;
   //    END_STRUCT;
   // END_VAR
BEGIN
END_DATA_BLOCK

DATA_BLOCK "iDB_ManageDoor"   // DB30
{ DB_Accessible_From_OPC_UA := 'FALSE' }
// stored: AutoNumber false, DBAccessibleFromOPCUA false, DBAccessibleFromWebserver false, InstanceOfName FB_ManageDoor, InstanceOfType FB
"FB_ManageDoor"
BEGIN
END_DATA_BLOCK

DATA_BLOCK "iDB_CommLeftRobot"   // DB401
{ DB_Accessible_From_OPC_UA := 'FALSE' }
// stored: AutoNumber false, DBAccessibleFromOPCUA false, DBAccessibleFromWebserver false, InstanceOfName FB40_CommSlave, InstanceOfType FB
"FB40_CommSlave"
BEGIN
END_DATA_BLOCK

DATA_BLOCK "iDB_CommRightRobot"   // DB402
{ DB_Accessible_From_OPC_UA := 'FALSE' }
// stored: AutoNumber false, DBAccessibleFromOPCUA false, DBAccessibleFromWebserver false, InstanceOfName FB40_CommSlave, InstanceOfType FB
"FB40_CommSlave"
BEGIN
END_DATA_BLOCK

DATA_BLOCK "iDB_ManageRecipe"   // DB55
{ DB_Accessible_From_OPC_UA := 'FALSE' }
// stored: AutoNumber false, DBAccessibleFromOPCUA false, DBAccessibleFromWebserver false, InstanceOfName FB50_ManageRecipe, InstanceOfType FB
"FB50_ManageRecipe"
BEGIN
END_DATA_BLOCK

DATA_BLOCK "iDB_FlatnessCtrlRecordLRobot"   // DB711
{ DB_Accessible_From_OPC_UA := 'FALSE' }
// stored: AutoNumber false, DBAccessibleFromOPCUA false, DBAccessibleFromWebserver false, InstanceOfName FB71_FlatnessCtrlRecord, InstanceOfType FB
"FB71_FlatnessCtrlRecord"
BEGIN
END_DATA_BLOCK

DATA_BLOCK "iDB_FlatnessCtrlRecordRRobot"   // DB712
{ DB_Accessible_From_OPC_UA := 'FALSE' }
// stored: AutoNumber false, DBAccessibleFromOPCUA false, DBAccessibleFromWebserver false, InstanceOfName FB71_FlatnessCtrlRecord, InstanceOfType FB
"FB71_FlatnessCtrlRecord"
BEGIN
END_DATA_BLOCK

DATA_BLOCK "iDB_ProductionRecord"   // DB700
{ DB_Accessible_From_OPC_UA := 'FALSE' }
// stored: AutoNumber false, DBAccessibleFromOPCUA false, DBAccessibleFromWebserver false, InstanceOfName FB70_ProductionRecord, InstanceOfType FB
"FB70_ProductionRecord"
BEGIN
END_DATA_BLOCK

DATA_BLOCK "iDB_TeepTrackRobot1"   // DB80
{ DB_Accessible_From_OPC_UA := 'FALSE' }
// stored: AutoNumber false, DBAccessibleFromOPCUA false, DBAccessibleFromWebserver false, InstanceOfName FB80_TeepTrack, InstanceOfType FB
"FB80_TeepTrack"
BEGIN
END_DATA_BLOCK

DATA_BLOCK "iDB_TeepTrackRobot2"   // DB81
// stored: AutoNumber false, InstanceOfName FB80_TeepTrack, InstanceOfType FB
"FB80_TeepTrack"
BEGIN
END_DATA_BLOCK

DATA_BLOCK "iDB_ReadPAC3200LeftRobot"   // DB91
{ DB_Accessible_From_OPC_UA := 'FALSE' }
// stored: AutoNumber false, DBAccessibleFromOPCUA false, DBAccessibleFromWebserver false, InstanceOfName FB_ReadSentronPAC3200, InstanceOfType FB
"FB_ReadSentronPAC3200"
BEGIN
END_DATA_BLOCK

DATA_BLOCK "iDB_ReadPAC3200MainPanel"   // DB90
{ DB_Accessible_From_OPC_UA := 'FALSE' }
// stored: AutoNumber false, DBAccessibleFromOPCUA false, DBAccessibleFromWebserver false, InstanceOfName FB_ReadSentronPAC3200, InstanceOfType FB
"FB_ReadSentronPAC3200"
BEGIN
END_DATA_BLOCK

DATA_BLOCK "iDB_ReadPAC3200RightRobot"   // DB92
{ DB_Accessible_From_OPC_UA := 'FALSE' }
// stored: AutoNumber false, DBAccessibleFromOPCUA false, DBAccessibleFromWebserver false, InstanceOfName FB_ReadSentronPAC3200, InstanceOfType FB
"FB_ReadSentronPAC3200"
BEGIN
END_DATA_BLOCK

DATA_BLOCK "iDBF_CaptiveKeyInLock"   // DB932, F_DB
{ DB_Accessible_From_OPC_UA := 'FALSE' }
// stored: AutoNumber false, DBAccessibleFromOPCUA false, DBAccessibleFromWebserver false, InstanceOfName EmergencyStop, InstanceOfType FB
"EmergencyStop"
   // VAR_INPUT
   //    xInputSafety { ExternalAccessible := 'False'; ExternalVisible := 'False'; ExternalWritable := 'False'} : Bool;
   //    xStateInput { ExternalAccessible := 'False'; ExternalVisible := 'False'; ExternalWritable := 'False'} : Bool;
   //    xAck { ExternalAccessible := 'False'; ExternalVisible := 'False'; ExternalWritable := 'False'} : Bool;
   //    xAllowAck { ExternalAccessible := 'False'; ExternalVisible := 'False'; ExternalWritable := 'False'} : Bool;
   // END_VAR
   // VAR_OUTPUT
   //    xStateSafety { ExternalAccessible := 'False'; ExternalVisible := 'False'; ExternalWritable := 'False'} : Bool;
   //    stSafetyState { ExternalAccessible := 'False'; ExternalVisible := 'False'; ExternalWritable := 'False'} : "stSafetyState";
   // END_VAR
   // VAR
   //    sx_Ack { ExternalAccessible := 'False'; ExternalVisible := 'False'; ExternalWritable := 'False'} : Bool;
   //    sx_TempAck { ExternalAccessible := 'False'; ExternalVisible := 'False'; ExternalWritable := 'False'} : Bool;
   //    sx_TempAckReq { ExternalAccessible := 'False'; ExternalVisible := 'False'; ExternalWritable := 'False'} : Bool;
   //    miDBF_EStop { ExternalAccessible := 'False'; ExternalVisible := 'False'; ExternalWritable := 'False'} : ESTOP1;
   // END_VAR
BEGIN
END_DATA_BLOCK

DATA_BLOCK "iDBF_DoorAcces"   // DB927, F_DB
{ DB_Accessible_From_OPC_UA := 'FALSE' }
// stored: AutoNumber false, DBAccessibleFromOPCUA false, DBAccessibleFromWebserver false, InstanceOfName GuardLocking, InstanceOfType FB
"GuardLocking"
   // VAR_INPUT
   //    xInputSafety_1 { ExternalAccessible := 'False'; ExternalVisible := 'False'; ExternalWritable := 'False'} : Bool;
   //    xInputSafety_2 { ExternalAccessible := 'False'; ExternalVisible := 'False'; ExternalWritable := 'False'} : Bool;
   //    xStateInputSafety_1 { ExternalAccessible := 'False'; ExternalVisible := 'False'; ExternalWritable := 'False'} : Bool;
   //    xStateInputSafety_2 { ExternalAccessible := 'False'; ExternalVisible := 'False'; ExternalWritable := 'False'} : Bool;
   //    xAck { ExternalAccessible := 'False'; ExternalVisible := 'False'; ExternalWritable := 'False'} : Bool;
   //    xAllowAck { ExternalAccessible := 'False'; ExternalVisible := 'False'; ExternalWritable := 'False'} : Bool;
   // END_VAR
   // VAR_OUTPUT
   //    xStateSafety { ExternalAccessible := 'False'; ExternalVisible := 'False'; ExternalWritable := 'False'} : Bool;
   //    stSafetyState { ExternalAccessible := 'False'; ExternalVisible := 'False'; ExternalWritable := 'False'} : "stSafetyState";
   // END_VAR
   // VAR
   //    sx_Ack { ExternalAccessible := 'False'; ExternalVisible := 'False'; ExternalWritable := 'False'} : Bool;
   //    sx_TempAck { ExternalAccessible := 'False'; ExternalVisible := 'False'; ExternalWritable := 'False'} : Bool;
   //    sx_TempAckReq { ExternalAccessible := 'False'; ExternalVisible := 'False'; ExternalWritable := 'False'} : Bool;
   //    miDBF_Interverrouillage { ExternalAccessible := 'False'; ExternalVisible := 'False'; ExternalWritable := 'False'} : SFDOOR;
   // END_VAR
BEGIN
END_DATA_BLOCK

DATA_BLOCK "iDBF_EStopControlRoom"   // DB926, F_DB
{ DB_Accessible_From_OPC_UA := 'FALSE' }
// stored: AutoNumber false, DBAccessibleFromOPCUA false, DBAccessibleFromWebserver false, InstanceOfName EmergencyStop, InstanceOfType FB
"EmergencyStop"
   // VAR_INPUT
   //    xInputSafety { ExternalAccessible := 'False'; ExternalVisible := 'False'; ExternalWritable := 'False'} : Bool;
   //    xStateInput { ExternalAccessible := 'False'; ExternalVisible := 'False'; ExternalWritable := 'False'} : Bool;
   //    xAck { ExternalAccessible := 'False'; ExternalVisible := 'False'; ExternalWritable := 'False'} : Bool;
   //    xAllowAck { ExternalAccessible := 'False'; ExternalVisible := 'False'; ExternalWritable := 'False'} : Bool;
   // END_VAR
   // VAR_OUTPUT
   //    xStateSafety { ExternalAccessible := 'False'; ExternalVisible := 'False'; ExternalWritable := 'False'} : Bool;
   //    stSafetyState { ExternalAccessible := 'False'; ExternalVisible := 'False'; ExternalWritable := 'False'} : "stSafetyState";
   // END_VAR
   // VAR
   //    sx_Ack { ExternalAccessible := 'False'; ExternalVisible := 'False'; ExternalWritable := 'False'} : Bool;
   //    sx_TempAck { ExternalAccessible := 'False'; ExternalVisible := 'False'; ExternalWritable := 'False'} : Bool;
   //    sx_TempAckReq { ExternalAccessible := 'False'; ExternalVisible := 'False'; ExternalWritable := 'False'} : Bool;
   //    miDBF_EStop { ExternalAccessible := 'False'; ExternalVisible := 'False'; ExternalWritable := 'False'} : ESTOP1;
   // END_VAR
BEGIN
END_DATA_BLOCK

DATA_BLOCK "iDBF_EStopEntryDoor"   // DB924, F_DB
{ DB_Accessible_From_OPC_UA := 'FALSE' }
// stored: AutoNumber false, DBAccessibleFromOPCUA false, DBAccessibleFromWebserver false, InstanceOfName EmergencyStop, InstanceOfType FB
"EmergencyStop"
   // VAR_INPUT
   //    xInputSafety { ExternalAccessible := 'False'; ExternalVisible := 'False'; ExternalWritable := 'False'} : Bool;
   //    xStateInput { ExternalAccessible := 'False'; ExternalVisible := 'False'; ExternalWritable := 'False'} : Bool;
   //    xAck { ExternalAccessible := 'False'; ExternalVisible := 'False'; ExternalWritable := 'False'} : Bool;
   //    xAllowAck { ExternalAccessible := 'False'; ExternalVisible := 'False'; ExternalWritable := 'False'} : Bool;
   // END_VAR
   // VAR_OUTPUT
   //    xStateSafety { ExternalAccessible := 'False'; ExternalVisible := 'False'; ExternalWritable := 'False'} : Bool;
   //    stSafetyState { ExternalAccessible := 'False'; ExternalVisible := 'False'; ExternalWritable := 'False'} : "stSafetyState";
   // END_VAR
   // VAR
   //    sx_Ack { ExternalAccessible := 'False'; ExternalVisible := 'False'; ExternalWritable := 'False'} : Bool;
   //    sx_TempAck { ExternalAccessible := 'False'; ExternalVisible := 'False'; ExternalWritable := 'False'} : Bool;
   //    sx_TempAckReq { ExternalAccessible := 'False'; ExternalVisible := 'False'; ExternalWritable := 'False'} : Bool;
   //    miDBF_EStop { ExternalAccessible := 'False'; ExternalVisible := 'False'; ExternalWritable := 'False'} : ESTOP1;
   // END_VAR
BEGIN
END_DATA_BLOCK

